  PROC DrawPart35()
    MoveL Offs(pOrigin,222.80,334.80,0.00),v40,z0,tPen\WObj:=wPaper;
    MoveL Offs(pOrigin,222.80,334.80,0.00),v40,z0,tPen\WObj:=wPaper;
    MoveL Offs(pOrigin,222.80,334.16,0.00),v40,z0,tPen\WObj:=wPaper;
    MoveL Offs(pOrigin,222.38,333.74,0.00),v40,z0,tPen\WObj:=wPaper;
    MoveL Offs(pOrigin,221.10,333.52,0.00),v40,z0,tPen\WObj:=wPaper;
    MoveL Offs(pOrigin,221.10,333.52,0.00),v40,z0,tPen\WObj:=wPaper;
    MoveL Offs(pOrigin,220.46,332.75,0.00),v40,z0,tPen\WObj:=wPaper;
    MoveL Offs(pOrigin,214.73,331.54,0.00),v40,z0,tPen\WObj:=wPaper;
    MoveL Offs(pOrigin,212.18,329.84,0.00),v40,z0,tPen\WObj:=wPaper;
    MoveL Offs(pOrigin,210.69,329.49,0.00),v40,z0,tPen\WObj:=wPaper;
    MoveL Offs(pOrigin,210.69,329.49,0.00),v40,z0,tPen\WObj:=wPaper;
    MoveL Offs(pOrigin,209.84,328.57,0.00),v40,z0,tPen\WObj:=wPaper;
    MoveL Offs(pOrigin,206.86,327.36,0.00),v40,z0,tPen\WObj:=wPaper;
    MoveL Offs(pOrigin,206.86,327.36,0.00),v40,z0,tPen\WObj:=wPaper;
    MoveL Offs(pOrigin,207.07,328.42,0.00),v40,z0,tPen\WObj:=wPaper;
    MoveL Offs(pOrigin,209.84,330.55,0.00),v40,z0,tPen\WObj:=wPaper;
    MoveL Offs(pOrigin,209.84,330.55,0.00),v40,z0,tPen\WObj:=wPaper;
    MoveL Offs(pOrigin,210.69,329.49,0.00),v40,z0,tPen\WObj:=wPaper;
    MoveL Offs(pOrigin,210.26,329.06,0.00),v40,z0,tPen\WObj:=wPaper;
    MoveL Offs(pOrigin,210.69,329.49,0.00),v40,z0,tPen\WObj:=wPaper;
    MoveL Offs(pOrigin,210.26,329.06,0.00),v40,fine,tPen\WObj:=wPaper;
    MoveL Offs(pOrigin,210.26,329.06,6.00),v60,z5,tPen\WObj:=wPaper;
    MoveL Offs(pOrigin,209.84,330.55,6.00),vTravel,z5,tPen\WObj:=wPaper;
    MoveL Offs(pOrigin,209.84,330.55,0.00),v60,z0,tPen\WObj:=wPaper;
    MoveL Offs(pOrigin,210.90,332.04,0.00),v40,z0,tPen\WObj:=wPaper;
    MoveL Offs(pOrigin,210.90,332.04,0.00),v40,z0,tPen\WObj:=wPaper;
    MoveL Offs(pOrigin,214.30,333.67,0.00),v40,z0,tPen\WObj:=wPaper;
    MoveL Offs(pOrigin,215.36,333.74,0.00),v40,z0,tPen\WObj:=wPaper;
    MoveL Offs(pOrigin,215.36,333.74,0.00),v40,z0,tPen\WObj:=wPaper;
    MoveL Offs(pOrigin,216.00,333.10,0.00),v40,z0,tPen\WObj:=wPaper;
    MoveL Offs(pOrigin,217.91,333.31,0.00),v40,z0,tPen\WObj:=wPaper;
    MoveL Offs(pOrigin,218.76,333.74,0.00),v40,z0,tPen\WObj:=wPaper;
    MoveL Offs(pOrigin,221.10,333.52,0.00),v40,z0,tPen\WObj:=wPaper;
    MoveL Offs(pOrigin,222.16,333.52,0.00),v40,z0,tPen\WObj:=wPaper;
    MoveL Offs(pOrigin,222.80,332.75,0.00),v40,z0,tPen\WObj:=wPaper;
    MoveL Offs(pOrigin,224.93,332.46,0.00),v40,z0,tPen\WObj:=wPaper;
    MoveL Offs(pOrigin,225.35,331.83,0.00),v40,fine,tPen\WObj:=wPaper;
    MoveL Offs(pOrigin,225.35,331.83,6.00),v60,z5,tPen\WObj:=wPaper;
    MoveL Offs(pOrigin,226.62,331.19,6.00),vTravel,z5,tPen\WObj:=wPaper;
    MoveL Offs(pOrigin,226.62,331.19,0.00),v60,z0,tPen\WObj:=wPaper;
    MoveL Offs(pOrigin,225.35,331.47,0.00),v40,z0,tPen\WObj:=wPaper;
    MoveL Offs(pOrigin,223.86,331.19,0.00),v40,z0,tPen\WObj:=wPaper;
    MoveL Offs(pOrigin,223.86,331.19,0.00),v40,z0,tPen\WObj:=wPaper;
    MoveL Offs(pOrigin,222.38,331.61,0.00),v40,z0,tPen\WObj:=wPaper;
    MoveL Offs(pOrigin,219.40,331.40,0.00),v40,z0,tPen\WObj:=wPaper;
    MoveL Offs(pOrigin,217.70,331.68,0.00),v40,z0,tPen\WObj:=wPaper;
    MoveL Offs(pOrigin,217.49,332.04,0.00),v40,fine,tPen\WObj:=wPaper;
    MoveL Offs(pOrigin,217.49,332.04,6.00),v60,z5,tPen\WObj:=wPaper;
    MoveL Offs(pOrigin,215.79,331.61,6.00),vTravel,z5,tPen\WObj:=wPaper;
    MoveL Offs(pOrigin,215.79,331.61,0.00),v60,z0,tPen\WObj:=wPaper;
    MoveL Offs(pOrigin,215.86,330.98,0.00),v40,z0,tPen\WObj:=wPaper;
    MoveL Offs(pOrigin,216.21,330.76,0.00),v40,z0,tPen\WObj:=wPaper;
    MoveL Offs(pOrigin,219.61,330.55,0.00),v40,z0,tPen\WObj:=wPaper;
    MoveL Offs(pOrigin,223.44,329.06,0.00),v40,z0,tPen\WObj:=wPaper;
    MoveL Offs(pOrigin,224.71,329.06,0.00),v40,z0,tPen\WObj:=wPaper;
    MoveL Offs(pOrigin,224.71,329.06,0.00),v40,z0,tPen\WObj:=wPaper;
    MoveL Offs(pOrigin,223.86,331.19,0.00),v40,fine,tPen\WObj:=wPaper;
    MoveL Offs(pOrigin,223.86,331.19,6.00),v60,z5,tPen\WObj:=wPaper;
    MoveL Offs(pOrigin,226.62,331.19,6.00),vTravel,z5,tPen\WObj:=wPaper;
    MoveL Offs(pOrigin,226.62,331.19,0.00),v60,z0,tPen\WObj:=wPaper;
    MoveL Offs(pOrigin,227.90,331.61,0.00),v40,z0,tPen\WObj:=wPaper;
    MoveL Offs(pOrigin,229.81,331.19,0.00),v40,fine,tPen\WObj:=wPaper;
    MoveL Offs(pOrigin,229.81,331.19,6.00),v60,z5,tPen\WObj:=wPaper;
    MoveL Offs(pOrigin,230.45,329.27,6.00),vTravel,z5,tPen\WObj:=wPaper;
    MoveL Offs(pOrigin,230.45,329.27,0.00),v60,z0,tPen\WObj:=wPaper;
    MoveL Offs(pOrigin,230.02,329.70,0.00),v40,z0,tPen\WObj:=wPaper;
    MoveL Offs(pOrigin,230.45,329.27,0.00),v40,fine,tPen\WObj:=wPaper;
    MoveL Offs(pOrigin,230.45,329.27,6.00),v60,z5,tPen\WObj:=wPaper;
    MoveL Offs(pOrigin,232.36,329.27,6.00),vTravel,z5,tPen\WObj:=wPaper;
    MoveL Offs(pOrigin,232.36,329.27,0.00),v60,z0,tPen\WObj:=wPaper;
    MoveL Offs(pOrigin,232.15,329.70,0.00),v40,z0,tPen\WObj:=wPaper;
    MoveL Offs(pOrigin,232.36,329.27,0.00),v40,z0,tPen\WObj:=wPaper;
    MoveL Offs(pOrigin,233.21,329.91,0.00),v40,z0,tPen\WObj:=wPaper;
    MoveL Offs(pOrigin,232.79,330.55,0.00),v40,z0,tPen\WObj:=wPaper;
    MoveL Offs(pOrigin,233.21,329.91,0.00),v40,z0,tPen\WObj:=wPaper;
    MoveL Offs(pOrigin,233.64,329.06,0.00),v40,z0,tPen\WObj:=wPaper;
    MoveL Offs(pOrigin,233.43,329.49,0.00),v40,z0,tPen\WObj:=wPaper;
    MoveL Offs(pOrigin,233.64,329.06,0.00),v40,fine,tPen\WObj:=wPaper;
    MoveL Offs(pOrigin,233.64,329.06,6.00),v60,z5,tPen\WObj:=wPaper;
    MoveL Offs(pOrigin,232.57,324.60,6.00),vTravel,z5,tPen\WObj:=wPaper;
    MoveL Offs(pOrigin,232.57,324.60,0.00),v60,z0,tPen\WObj:=wPaper;
    MoveL Offs(pOrigin,232.79,325.02,0.00),v40,z0,tPen\WObj:=wPaper;
    MoveL Offs(pOrigin,232.57,324.60,0.00),v40,fine,tPen\WObj:=wPaper;
    MoveL Offs(pOrigin,232.57,324.60,6.00),v60,z5,tPen\WObj:=wPaper;
    MoveL Offs(pOrigin,231.94,323.54,6.00),vTravel,z5,tPen\WObj:=wPaper;
    MoveL Offs(pOrigin,231.94,323.54,0.00),v60,z0,tPen\WObj:=wPaper;
    MoveL Offs(pOrigin,232.36,324.17,0.00),v40,z0,tPen\WObj:=wPaper;
    MoveL Offs(pOrigin,231.94,323.54,0.00),v40,z0,tPen\WObj:=wPaper;
    MoveL Offs(pOrigin,231.09,323.33,0.00),v40,z0,tPen\WObj:=wPaper;
    MoveL Offs(pOrigin,228.54,319.71,0.00),v40,fine,tPen\WObj:=wPaper;
    MoveL Offs(pOrigin,228.54,319.71,6.00),v60,z5,tPen\WObj:=wPaper;
    MoveL Offs(pOrigin,228.54,318.23,6.00),vTravel,z5,tPen\WObj:=wPaper;
    MoveL Offs(pOrigin,228.54,318.23,0.00),v60,z0,tPen\WObj:=wPaper;
    MoveL Offs(pOrigin,226.84,314.40,0.00),v40,z0,tPen\WObj:=wPaper;
    MoveL Offs(pOrigin,226.84,313.12,0.00),v40,z0,tPen\WObj:=wPaper;
    MoveL Offs(pOrigin,227.48,310.65,0.00),v40,z0,tPen\WObj:=wPaper;
    MoveL Offs(pOrigin,225.42,310.79,0.00),v40,z0,tPen\WObj:=wPaper;
    MoveL Offs(pOrigin,224.64,312.49,0.00),v40,z0,tPen\WObj:=wPaper;
    MoveL Offs(pOrigin,224.64,313.76,0.00),v40,z0,tPen\WObj:=wPaper;
    MoveL Offs(pOrigin,224.07,314.61,0.00),v40,z0,tPen\WObj:=wPaper;
    MoveL Offs(pOrigin,224.29,316.10,0.00),v40,fine,tPen\WObj:=wPaper;
    MoveL Offs(pOrigin,224.29,316.10,6.00),v60,z5,tPen\WObj:=wPaper;
    MoveL Offs(pOrigin,223.86,313.76,6.00),vTravel,z5,tPen\WObj:=wPaper;
    MoveL Offs(pOrigin,223.86,313.76,0.00),v60,z0,tPen\WObj:=wPaper;
    MoveL Offs(pOrigin,223.86,313.34,0.00),v40,z0,tPen\WObj:=wPaper;
    MoveL Offs(pOrigin,224.50,312.91,0.00),v40,fine,tPen\WObj:=wPaper;
    MoveL Offs(pOrigin,224.50,312.91,6.00),v60,z5,tPen\WObj:=wPaper;
    MoveL Offs(pOrigin,223.01,313.76,6.00),vTravel,z5,tPen\WObj:=wPaper;
    MoveL Offs(pOrigin,223.01,313.76,0.00),v60,z0,tPen\WObj:=wPaper;
    MoveL Offs(pOrigin,222.59,314.61,0.00),v40,z0,tPen\WObj:=wPaper;
    MoveL Offs(pOrigin,222.38,316.52,0.00),v40,z0,tPen\WObj:=wPaper;
    MoveL Offs(pOrigin,221.60,316.95,0.00),v40,z0,tPen\WObj:=wPaper;
    MoveL Offs(pOrigin,221.52,317.59,0.00),v40,z0,tPen\WObj:=wPaper;
    MoveL Offs(pOrigin,223.30,320.35,0.00),v40,z0,tPen\WObj:=wPaper;
    MoveL Offs(pOrigin,224.07,322.48,0.00),v40,z0,tPen\WObj:=wPaper;
    MoveL Offs(pOrigin,224.07,322.48,0.00),v40,z0,tPen\WObj:=wPaper;
    MoveL Offs(pOrigin,224.78,323.11,0.00),v40,z0,tPen\WObj:=wPaper;
    MoveL Offs(pOrigin,225.14,324.17,0.00),v40,z0,tPen\WObj:=wPaper;
    MoveL Offs(pOrigin,224.93,327.79,0.00),v40,z0,tPen\WObj:=wPaper;
    MoveL Offs(pOrigin,224.93,328.21,0.00),v40,z0,tPen\WObj:=wPaper;
  ENDPROC

  PROC DrawPart36()
    MoveL Offs(pOrigin,225.70,327.15,0.00),v40,z0,tPen\WObj:=wPaper;
    MoveL Offs(pOrigin,226.20,325.24,0.00),v40,z0,tPen\WObj:=wPaper;
    MoveL Offs(pOrigin,225.63,321.62,0.00),v40,z0,tPen\WObj:=wPaper;
    MoveL Offs(pOrigin,225.99,321.55,0.00),v40,z0,tPen\WObj:=wPaper;
    MoveL Offs(pOrigin,227.33,323.54,0.00),v40,z0,tPen\WObj:=wPaper;
    MoveL Offs(pOrigin,227.90,326.51,0.00),v40,z0,tPen\WObj:=wPaper;
    MoveL Offs(pOrigin,227.26,327.72,0.00),v40,z0,tPen\WObj:=wPaper;
    MoveL Offs(pOrigin,225.35,328.64,0.00),v40,z0,tPen\WObj:=wPaper;
    MoveL Offs(pOrigin,224.93,328.21,0.00),v40,fine,tPen\WObj:=wPaper;
    MoveL Offs(pOrigin,224.93,328.21,6.00),v60,z5,tPen\WObj:=wPaper;
    MoveL Offs(pOrigin,227.05,328.00,6.00),vTravel,z5,tPen\WObj:=wPaper;
    MoveL Offs(pOrigin,227.05,328.00,0.00),v60,z0,tPen\WObj:=wPaper;
    MoveL Offs(pOrigin,227.26,327.58,0.00),v40,z0,tPen\WObj:=wPaper;
    MoveL Offs(pOrigin,227.05,328.00,0.00),v40,fine,tPen\WObj:=wPaper;
    MoveL Offs(pOrigin,227.05,328.00,6.00),v60,z5,tPen\WObj:=wPaper;
    MoveL Offs(pOrigin,227.90,326.30,6.00),vTravel,z5,tPen\WObj:=wPaper;
    MoveL Offs(pOrigin,227.90,326.30,0.00),v60,z0,tPen\WObj:=wPaper;
    MoveL Offs(pOrigin,228.54,325.66,0.00),v40,z0,tPen\WObj:=wPaper;
    MoveL Offs(pOrigin,228.32,322.26,0.00),v40,fine,tPen\WObj:=wPaper;
    MoveL Offs(pOrigin,228.32,322.26,6.00),v60,z5,tPen\WObj:=wPaper;
    MoveL Offs(pOrigin,226.41,321.62,6.00),vTravel,z5,tPen\WObj:=wPaper;
    MoveL Offs(pOrigin,226.41,321.62,0.00),v60,z0,tPen\WObj:=wPaper;
    MoveL Offs(pOrigin,226.62,322.05,0.00),v40,z0,tPen\WObj:=wPaper;
    MoveL Offs(pOrigin,226.41,321.62,0.00),v40,z0,tPen\WObj:=wPaper;
    MoveL Offs(pOrigin,225.56,321.41,0.00),v40,z0,tPen\WObj:=wPaper;
    MoveL Offs(pOrigin,224.07,318.86,0.00),v40,fine,tPen\WObj:=wPaper;
    MoveL Offs(pOrigin,224.07,318.86,6.00),v60,z5,tPen\WObj:=wPaper;
    MoveL Offs(pOrigin,224.07,322.48,6.00),vTravel,z5,tPen\WObj:=wPaper;
    MoveL Offs(pOrigin,224.07,322.48,0.00),v60,z0,tPen\WObj:=wPaper;
    MoveL Offs(pOrigin,223.37,326.09,0.00),v40,z0,tPen\WObj:=wPaper;
    MoveL Offs(pOrigin,221.95,327.65,0.00),v40,z0,tPen\WObj:=wPaper;
    MoveL Offs(pOrigin,217.91,329.27,0.00),v40,z0,tPen\WObj:=wPaper;
    MoveL Offs(pOrigin,215.57,329.49,0.00),v40,z0,tPen\WObj:=wPaper;
    MoveL Offs(pOrigin,213.45,329.27,0.00),v40,z0,tPen\WObj:=wPaper;
    MoveL Offs(pOrigin,212.60,329.91,0.00),v40,fine,tPen\WObj:=wPaper;
    MoveL Offs(pOrigin,212.60,329.91,6.00),v60,z5,tPen\WObj:=wPaper;
    MoveL Offs(pOrigin,214.51,330.98,6.00),vTravel,z5,tPen\WObj:=wPaper;
    MoveL Offs(pOrigin,214.51,330.98,0.00),v60,z0,tPen\WObj:=wPaper;
    MoveL Offs(pOrigin,214.94,330.55,0.00),v40,z0,tPen\WObj:=wPaper;
    MoveL Offs(pOrigin,215.79,330.76,0.00),v40,fine,tPen\WObj:=wPaper;
    MoveL Offs(pOrigin,215.79,330.76,6.00),v60,z5,tPen\WObj:=wPaper;
    MoveL Offs(pOrigin,215.36,333.74,6.00),vTravel,z5,tPen\WObj:=wPaper;
    MoveL Offs(pOrigin,215.36,333.74,0.00),v60,z0,tPen\WObj:=wPaper;
    MoveL Offs(pOrigin,216.43,334.16,0.00),v40,z0,tPen\WObj:=wPaper;
    MoveL Offs(pOrigin,218.12,334.16,0.00),v40,z0,tPen\WObj:=wPaper;
    MoveL Offs(pOrigin,218.34,333.74,0.00),v40,fine,tPen\WObj:=wPaper;
    MoveL Offs(pOrigin,218.34,333.74,6.00),v60,z5,tPen\WObj:=wPaper;
    MoveL Offs(pOrigin,217.91,335.23,6.00),vTravel,z5,tPen\WObj:=wPaper;
    MoveL Offs(pOrigin,217.91,335.23,0.00),v60,z0,tPen\WObj:=wPaper;
    MoveL Offs(pOrigin,221.95,335.86,0.00),v40,z0,tPen\WObj:=wPaper;
    MoveL Offs(pOrigin,221.95,335.86,0.00),v40,z0,tPen\WObj:=wPaper;
    MoveL Offs(pOrigin,222.02,336.29,0.00),v40,z0,tPen\WObj:=wPaper;
    MoveL Offs(pOrigin,222.80,336.71,0.00),v40,z0,tPen\WObj:=wPaper;
    MoveL Offs(pOrigin,225.99,336.92,0.00),v40,z0,tPen\WObj:=wPaper;
    MoveL Offs(pOrigin,225.99,336.92,0.00),v40,z0,tPen\WObj:=wPaper;
    MoveL Offs(pOrigin,226.84,337.35,0.00),v40,fine,tPen\WObj:=wPaper;
    MoveL Offs(pOrigin,226.84,337.35,6.00),v60,z5,tPen\WObj:=wPaper;
    MoveL Offs(pOrigin,224.71,335.86,6.00),vTravel,z5,tPen\WObj:=wPaper;
    MoveL Offs(pOrigin,224.71,335.86,0.00),v60,z0,tPen\WObj:=wPaper;
    MoveL Offs(pOrigin,222.59,335.65,0.00),v40,fine,tPen\WObj:=wPaper;
    MoveL Offs(pOrigin,222.59,335.65,6.00),v60,z5,tPen\WObj:=wPaper;
    MoveL Offs(pOrigin,226.62,331.19,6.00),vTravel,z5,tPen\WObj:=wPaper;
    MoveL Offs(pOrigin,226.62,331.19,0.00),v60,z0,tPen\WObj:=wPaper;
    MoveL Offs(pOrigin,229.53,328.64,0.00),v40,z0,tPen\WObj:=wPaper;
    MoveL Offs(pOrigin,230.02,327.36,0.00),v40,z0,tPen\WObj:=wPaper;
    MoveL Offs(pOrigin,230.02,325.02,0.00),v40,z0,tPen\WObj:=wPaper;
    MoveL Offs(pOrigin,229.10,322.55,0.00),v40,z0,tPen\WObj:=wPaper;
    MoveL Offs(pOrigin,228.32,322.05,0.00),v40,z0,tPen\WObj:=wPaper;
    MoveL Offs(pOrigin,226.13,318.65,0.00),v40,z0,tPen\WObj:=wPaper;
    MoveL Offs(pOrigin,225.70,316.95,0.00),v40,z0,tPen\WObj:=wPaper;
    MoveL Offs(pOrigin,226.41,316.31,0.00),v40,z0,tPen\WObj:=wPaper;
    MoveL Offs(pOrigin,225.99,315.25,0.00),v40,z0,tPen\WObj:=wPaper;
    MoveL Offs(pOrigin,226.20,314.61,0.00),v40,z0,tPen\WObj:=wPaper;
    MoveL Offs(pOrigin,227.05,314.61,0.00),v40,z0,tPen\WObj:=wPaper;
    MoveL Offs(pOrigin,228.18,312.13,0.00),v40,z0,tPen\WObj:=wPaper;
    MoveL Offs(pOrigin,228.96,311.85,0.00),v40,z0,tPen\WObj:=wPaper;
    MoveL Offs(pOrigin,228.96,311.85,0.00),v40,z0,tPen\WObj:=wPaper;
    MoveL Offs(pOrigin,229.39,311.00,0.00),v40,z0,tPen\WObj:=wPaper;
    MoveL Offs(pOrigin,229.39,311.00,0.00),v40,z0,tPen\WObj:=wPaper;
    MoveL Offs(pOrigin,228.54,310.15,0.00),v40,z0,tPen\WObj:=wPaper;
    MoveL Offs(pOrigin,227.69,310.58,0.00),v40,z0,tPen\WObj:=wPaper;
    MoveL Offs(pOrigin,228.75,310.15,0.00),v40,z0,tPen\WObj:=wPaper;
    MoveL Offs(pOrigin,229.39,311.00,0.00),v40,z0,tPen\WObj:=wPaper;
    MoveL Offs(pOrigin,229.39,311.00,0.00),v40,z0,tPen\WObj:=wPaper;
    MoveL Offs(pOrigin,230.02,311.00,0.00),v40,z0,tPen\WObj:=wPaper;
    MoveL Offs(pOrigin,230.88,312.06,0.00),v40,z0,tPen\WObj:=wPaper;
    MoveL Offs(pOrigin,230.88,311.64,0.00),v40,z0,tPen\WObj:=wPaper;
    MoveL Offs(pOrigin,232.57,310.58,0.00),v40,z0,tPen\WObj:=wPaper;
    MoveL Offs(pOrigin,233.43,311.00,0.00),v40,fine,tPen\WObj:=wPaper;
    MoveL Offs(pOrigin,233.43,311.00,6.00),v60,z5,tPen\WObj:=wPaper;
    MoveL Offs(pOrigin,235.55,311.42,6.00),vTravel,z5,tPen\WObj:=wPaper;
    MoveL Offs(pOrigin,235.55,311.42,0.00),v60,z0,tPen\WObj:=wPaper;
    MoveL Offs(pOrigin,234.98,311.71,0.00),v40,z0,tPen\WObj:=wPaper;
    MoveL Offs(pOrigin,234.70,312.49,0.00),v40,z0,tPen\WObj:=wPaper;
    MoveL Offs(pOrigin,234.70,315.46,0.00),v40,z0,tPen\WObj:=wPaper;
    MoveL Offs(pOrigin,235.12,317.38,0.00),v40,fine,tPen\WObj:=wPaper;
    MoveL Offs(pOrigin,235.12,317.38,6.00),v60,z5,tPen\WObj:=wPaper;
    MoveL Offs(pOrigin,232.79,318.44,6.00),vTravel,z5,tPen\WObj:=wPaper;
    MoveL Offs(pOrigin,232.79,318.44,0.00),v60,z0,tPen\WObj:=wPaper;
    MoveL Offs(pOrigin,234.27,320.14,0.00),v40,z0,tPen\WObj:=wPaper;
    MoveL Offs(pOrigin,234.27,320.56,0.00),v40,fine,tPen\WObj:=wPaper;
    MoveL Offs(pOrigin,234.27,320.56,6.00),v60,z5,tPen\WObj:=wPaper;
    MoveL Offs(pOrigin,235.55,321.41,6.00),vTravel,z5,tPen\WObj:=wPaper;
    MoveL Offs(pOrigin,235.55,321.41,0.00),v60,z0,tPen\WObj:=wPaper;
    MoveL Offs(pOrigin,234.91,320.70,0.00),v40,z0,tPen\WObj:=wPaper;
    MoveL Offs(pOrigin,234.35,320.77,0.00),v40,z0,tPen\WObj:=wPaper;
    MoveL Offs(pOrigin,234.70,321.84,0.00),v40,z0,tPen\WObj:=wPaper;
    MoveL Offs(pOrigin,235.55,322.05,0.00),v40,z0,tPen\WObj:=wPaper;
    MoveL Offs(pOrigin,235.55,322.05,0.00),v40,z0,tPen\WObj:=wPaper;
    MoveL Offs(pOrigin,237.89,325.66,0.00),v40,fine,tPen\WObj:=wPaper;
    MoveL Offs(pOrigin,237.89,325.66,6.00),v60,z5,tPen\WObj:=wPaper;
    MoveL Offs(pOrigin,239.80,326.73,6.00),vTravel,z5,tPen\WObj:=wPaper;
    MoveL Offs(pOrigin,239.80,326.73,0.00),v60,z0,tPen\WObj:=wPaper;
    MoveL Offs(pOrigin,239.16,327.15,0.00),v40,z0,tPen\WObj:=wPaper;
    MoveL Offs(pOrigin,239.38,328.00,0.00),v40,fine,tPen\WObj:=wPaper;
    MoveL Offs(pOrigin,239.38,328.00,6.00),v60,z5,tPen\WObj:=wPaper;
    MoveL Offs(pOrigin,242.14,324.60,6.00),vTravel,z5,tPen\WObj:=wPaper;
    MoveL Offs(pOrigin,242.14,324.60,0.00),v60,z0,tPen\WObj:=wPaper;
    MoveL Offs(pOrigin,242.56,325.24,0.00),v40,z0,tPen\WObj:=wPaper;
    MoveL Offs(pOrigin,242.14,324.60,0.00),v40,fine,tPen\WObj:=wPaper;
  ENDPROC

  PROC DrawPart37()
    MoveL Offs(pOrigin,242.14,324.60,6.00),v60,z5,tPen\WObj:=wPaper;
    MoveL Offs(pOrigin,239.59,323.11,6.00),vTravel,z5,tPen\WObj:=wPaper;
    MoveL Offs(pOrigin,239.59,323.11,0.00),v60,z0,tPen\WObj:=wPaper;
    MoveL Offs(pOrigin,237.04,320.77,0.00),v40,z0,tPen\WObj:=wPaper;
    MoveL Offs(pOrigin,237.04,320.77,0.00),v40,z0,tPen\WObj:=wPaper;
    MoveL Offs(pOrigin,235.76,321.41,0.00),v40,z0,tPen\WObj:=wPaper;
    MoveL Offs(pOrigin,235.55,322.05,0.00),v40,fine,tPen\WObj:=wPaper;
    MoveL Offs(pOrigin,235.55,322.05,6.00),v60,z5,tPen\WObj:=wPaper;
    MoveL Offs(pOrigin,237.04,320.77,6.00),vTravel,z5,tPen\WObj:=wPaper;
    MoveL Offs(pOrigin,237.04,320.77,0.00),v60,z0,tPen\WObj:=wPaper;
    MoveL Offs(pOrigin,235.34,317.80,0.00),v40,z0,tPen\WObj:=wPaper;
    MoveL Offs(pOrigin,234.20,316.95,0.00),v40,z0,tPen\WObj:=wPaper;
    MoveL Offs(pOrigin,233.64,315.25,0.00),v40,z0,tPen\WObj:=wPaper;
    MoveL Offs(pOrigin,233.43,313.34,0.00),v40,z0,tPen\WObj:=wPaper;
    MoveL Offs(pOrigin,233.64,312.49,0.00),v40,z0,tPen\WObj:=wPaper;
    MoveL Offs(pOrigin,233.21,311.99,0.00),v40,z0,tPen\WObj:=wPaper;
    MoveL Offs(pOrigin,232.57,313.12,0.00),v40,z0,tPen\WObj:=wPaper;
    MoveL Offs(pOrigin,232.57,315.25,0.00),v40,z0,tPen\WObj:=wPaper;
    MoveL Offs(pOrigin,233.21,317.16,0.00),v40,z0,tPen\WObj:=wPaper;
    MoveL Offs(pOrigin,232.79,318.44,0.00),v40,z0,tPen\WObj:=wPaper;
    MoveL Offs(pOrigin,232.79,318.44,0.00),v40,z0,tPen\WObj:=wPaper;
    MoveL Offs(pOrigin,232.15,317.80,0.00),v40,z0,tPen\WObj:=wPaper;
    MoveL Offs(pOrigin,232.15,317.80,0.00),v40,z0,tPen\WObj:=wPaper;
    MoveL Offs(pOrigin,231.51,314.61,0.00),v40,z0,tPen\WObj:=wPaper;
    MoveL Offs(pOrigin,230.88,313.76,0.00),v40,z0,tPen\WObj:=wPaper;
    MoveL Offs(pOrigin,230.88,313.76,0.00),v40,z0,tPen\WObj:=wPaper;
    MoveL Offs(pOrigin,230.80,312.27,0.00),v40,z0,tPen\WObj:=wPaper;
    MoveL Offs(pOrigin,229.25,312.91,0.00),v40,z0,tPen\WObj:=wPaper;
    MoveL Offs(pOrigin,228.96,316.74,0.00),v40,z0,tPen\WObj:=wPaper;
    MoveL Offs(pOrigin,228.96,316.74,0.00),v40,z0,tPen\WObj:=wPaper;
    MoveL Offs(pOrigin,229.81,316.74,0.00),v40,z0,tPen\WObj:=wPaper;
    MoveL Offs(pOrigin,230.66,318.01,0.00),v40,z0,tPen\WObj:=wPaper;
    MoveL Offs(pOrigin,230.66,318.01,0.00),v40,z0,tPen\WObj:=wPaper;
    MoveL Offs(pOrigin,231.09,319.08,0.00),v40,z0,tPen\WObj:=wPaper;
    MoveL Offs(pOrigin,231.09,319.08,0.00),v40,z0,tPen\WObj:=wPaper;
    MoveL Offs(pOrigin,231.16,320.56,0.00),v40,z0,tPen\WObj:=wPaper;
    MoveL Offs(pOrigin,233.43,323.11,0.00),v40,z0,tPen\WObj:=wPaper;
    MoveL Offs(pOrigin,233.21,322.69,0.00),v40,z0,tPen\WObj:=wPaper;
    MoveL Offs(pOrigin,233.43,323.11,0.00),v40,z0,tPen\WObj:=wPaper;
    MoveL Offs(pOrigin,233.21,322.69,0.00),v40,fine,tPen\WObj:=wPaper;
    MoveL Offs(pOrigin,233.21,322.69,6.00),v60,z5,tPen\WObj:=wPaper;
    MoveL Offs(pOrigin,231.09,319.08,6.00),vTravel,z5,tPen\WObj:=wPaper;
    MoveL Offs(pOrigin,231.09,319.08,0.00),v60,z0,tPen\WObj:=wPaper;
    MoveL Offs(pOrigin,231.94,319.08,0.00),v40,z0,tPen\WObj:=wPaper;
    MoveL Offs(pOrigin,232.57,318.44,0.00),v40,z0,tPen\WObj:=wPaper;
    MoveL Offs(pOrigin,232.57,318.44,0.00),v40,z0,tPen\WObj:=wPaper;
    MoveL Offs(pOrigin,231.94,317.80,0.00),v40,z0,tPen\WObj:=wPaper;
    MoveL Offs(pOrigin,231.30,317.80,0.00),v40,z0,tPen\WObj:=wPaper;
    MoveL Offs(pOrigin,231.30,317.80,0.00),v40,z0,tPen\WObj:=wPaper;
    MoveL Offs(pOrigin,231.09,316.52,0.00),v40,z0,tPen\WObj:=wPaper;
    MoveL Offs(pOrigin,230.45,316.10,0.00),v40,z0,tPen\WObj:=wPaper;
    MoveL Offs(pOrigin,230.45,316.10,0.00),v40,z0,tPen\WObj:=wPaper;
    MoveL Offs(pOrigin,230.45,314.19,0.00),v40,z0,tPen\WObj:=wPaper;
    MoveL Offs(pOrigin,230.88,313.76,0.00),v40,fine,tPen\WObj:=wPaper;
    MoveL Offs(pOrigin,230.88,313.76,6.00),v60,z5,tPen\WObj:=wPaper;
    MoveL Offs(pOrigin,230.88,311.64,6.00),vTravel,z5,tPen\WObj:=wPaper;
    MoveL Offs(pOrigin,230.88,311.64,0.00),v60,z0,tPen\WObj:=wPaper;
    MoveL Offs(pOrigin,230.24,311.00,0.00),v40,fine,tPen\WObj:=wPaper;
    MoveL Offs(pOrigin,230.24,311.00,6.00),v60,z5,tPen\WObj:=wPaper;
    MoveL Offs(pOrigin,226.84,309.30,6.00),vTravel,z5,tPen\WObj:=wPaper;
    MoveL Offs(pOrigin,226.84,309.30,0.00),v60,z0,tPen\WObj:=wPaper;
    MoveL Offs(pOrigin,225.56,310.36,0.00),v40,z0,tPen\WObj:=wPaper;
    MoveL Offs(pOrigin,224.07,310.15,0.00),v40,z0,tPen\WObj:=wPaper;
    MoveL Offs(pOrigin,222.59,310.50,0.00),v40,z0,tPen\WObj:=wPaper;
    MoveL Offs(pOrigin,222.45,309.51,0.00),v40,z0,tPen\WObj:=wPaper;
    MoveL Offs(pOrigin,223.86,308.88,0.00),v40,fine,tPen\WObj:=wPaper;
    MoveL Offs(pOrigin,223.86,308.88,6.00),v60,z5,tPen\WObj:=wPaper;
    MoveL Offs(pOrigin,222.38,309.30,6.00),vTravel,z5,tPen\WObj:=wPaper;
    MoveL Offs(pOrigin,222.38,309.30,0.00),v60,z0,tPen\WObj:=wPaper;
    MoveL Offs(pOrigin,221.31,308.66,0.00),v40,z0,tPen\WObj:=wPaper;
    MoveL Offs(pOrigin,220.89,308.88,0.00),v40,z0,tPen\WObj:=wPaper;
    MoveL Offs(pOrigin,220.46,308.24,0.00),v40,z0,tPen\WObj:=wPaper;
    MoveL Offs(pOrigin,220.46,308.24,0.00),v40,z0,tPen\WObj:=wPaper;
    MoveL Offs(pOrigin,220.68,308.24,0.00),v40,z0,tPen\WObj:=wPaper;
    MoveL Offs(pOrigin,220.04,307.39,0.00),v40,z0,tPen\WObj:=wPaper;
    MoveL Offs(pOrigin,218.76,307.39,0.00),v40,z0,tPen\WObj:=wPaper;
    MoveL Offs(pOrigin,218.76,307.39,0.00),v40,z0,tPen\WObj:=wPaper;
    MoveL Offs(pOrigin,218.12,306.61,0.00),v40,z0,tPen\WObj:=wPaper;
    MoveL Offs(pOrigin,217.06,306.61,0.00),v40,z0,tPen\WObj:=wPaper;
    MoveL Offs(pOrigin,217.49,308.02,0.00),v40,z0,tPen\WObj:=wPaper;
    MoveL Offs(pOrigin,217.49,308.02,0.00),v40,z0,tPen\WObj:=wPaper;
    MoveL Offs(pOrigin,218.34,308.02,0.00),v40,z0,tPen\WObj:=wPaper;
    MoveL Offs(pOrigin,218.76,308.45,0.00),v40,z0,tPen\WObj:=wPaper;
    MoveL Offs(pOrigin,218.76,309.51,0.00),v40,z0,tPen\WObj:=wPaper;
    MoveL Offs(pOrigin,218.76,309.51,0.00),v40,z0,tPen\WObj:=wPaper;
    MoveL Offs(pOrigin,220.68,309.09,0.00),v40,z0,tPen\WObj:=wPaper;
    MoveL Offs(pOrigin,220.46,308.24,0.00),v40,z0,tPen\WObj:=wPaper;
    MoveL Offs(pOrigin,218.76,308.24,0.00),v40,fine,tPen\WObj:=wPaper;
    MoveL Offs(pOrigin,218.76,308.24,6.00),v60,z5,tPen\WObj:=wPaper;
    MoveL Offs(pOrigin,217.49,308.02,6.00),vTravel,z5,tPen\WObj:=wPaper;
    MoveL Offs(pOrigin,217.49,308.02,0.00),v60,z0,tPen\WObj:=wPaper;
    MoveL Offs(pOrigin,215.79,308.45,0.00),v40,z0,tPen\WObj:=wPaper;
    MoveL Offs(pOrigin,214.94,309.16,0.00),v40,z0,tPen\WObj:=wPaper;
    MoveL Offs(pOrigin,214.51,308.88,0.00),v40,z0,tPen\WObj:=wPaper;
    MoveL Offs(pOrigin,214.73,309.30,0.00),v40,z0,tPen\WObj:=wPaper;
    MoveL Offs(pOrigin,214.09,308.52,0.00),v40,z0,tPen\WObj:=wPaper;
    MoveL Offs(pOrigin,213.45,308.38,0.00),v40,z0,tPen\WObj:=wPaper;
    MoveL Offs(pOrigin,210.26,309.94,0.00),v40,z0,tPen\WObj:=wPaper;
    MoveL Offs(pOrigin,210.26,309.94,0.00),v40,z0,tPen\WObj:=wPaper;
    MoveL Offs(pOrigin,209.98,310.72,0.00),v40,z0,tPen\WObj:=wPaper;
    MoveL Offs(pOrigin,207.50,312.27,0.00),v40,z0,tPen\WObj:=wPaper;
    MoveL Offs(pOrigin,206.65,313.55,0.00),v40,z0,tPen\WObj:=wPaper;
    MoveL Offs(pOrigin,206.65,313.55,0.00),v40,z0,tPen\WObj:=wPaper;
    MoveL Offs(pOrigin,206.44,313.98,0.00),v40,z0,tPen\WObj:=wPaper;
    MoveL Offs(pOrigin,205.16,314.40,0.00),v40,z0,tPen\WObj:=wPaper;
    MoveL Offs(pOrigin,205.16,314.40,0.00),v40,z0,tPen\WObj:=wPaper;
    MoveL Offs(pOrigin,204.31,314.19,0.00),v40,z0,tPen\WObj:=wPaper;
    MoveL Offs(pOrigin,203.89,314.61,0.00),v40,z0,tPen\WObj:=wPaper;
    MoveL Offs(pOrigin,203.89,314.61,0.00),v40,z0,tPen\WObj:=wPaper;
    MoveL Offs(pOrigin,202.19,314.40,0.00),v40,z0,tPen\WObj:=wPaper;
    MoveL Offs(pOrigin,201.76,315.04,0.00),v40,fine,tPen\WObj:=wPaper;
    MoveL Offs(pOrigin,201.76,315.04,6.00),v60,z5,tPen\WObj:=wPaper;
    MoveL Offs(pOrigin,203.04,315.67,6.00),vTravel,z5,tPen\WObj:=wPaper;
    MoveL Offs(pOrigin,203.04,315.67,0.00),v60,z0,tPen\WObj:=wPaper;
    MoveL Offs(pOrigin,203.46,316.10,0.00),v40,z0,tPen\WObj:=wPaper;
    MoveL Offs(pOrigin,205.38,316.10,0.00),v40,z0,tPen\WObj:=wPaper;
    MoveL Offs(pOrigin,205.38,316.10,0.00),v40,z0,tPen\WObj:=wPaper;
    MoveL Offs(pOrigin,205.59,316.88,0.00),v40,z0,tPen\WObj:=wPaper;
    MoveL Offs(pOrigin,206.86,316.95,0.00),v40,z0,tPen\WObj:=wPaper;
    MoveL Offs(pOrigin,208.35,316.52,0.00),v40,z0,tPen\WObj:=wPaper;
  ENDPROC

  PROC DrawPart38()
    MoveL Offs(pOrigin,209.41,316.60,0.00),v40,z0,tPen\WObj:=wPaper;
    MoveL Offs(pOrigin,210.69,315.75,0.00),v40,z0,tPen\WObj:=wPaper;
    MoveL Offs(pOrigin,211.32,315.67,0.00),v40,z0,tPen\WObj:=wPaper;
    MoveL Offs(pOrigin,211.32,315.67,0.00),v40,z0,tPen\WObj:=wPaper;
    MoveL Offs(pOrigin,211.96,315.89,0.00),v40,z0,tPen\WObj:=wPaper;
    MoveL Offs(pOrigin,212.18,316.74,0.00),v40,z0,tPen\WObj:=wPaper;
    MoveL Offs(pOrigin,211.68,318.65,0.00),v40,z0,tPen\WObj:=wPaper;
    MoveL Offs(pOrigin,210.90,319.71,0.00),v40,z0,tPen\WObj:=wPaper;
    MoveL Offs(pOrigin,210.90,319.71,0.00),v40,z0,tPen\WObj:=wPaper;
    MoveL Offs(pOrigin,211.96,320.99,0.00),v40,z0,tPen\WObj:=wPaper;
    MoveL Offs(pOrigin,211.96,320.99,0.00),v40,z0,tPen\WObj:=wPaper;
    MoveL Offs(pOrigin,213.10,320.35,0.00),v40,z0,tPen\WObj:=wPaper;
    MoveL Offs(pOrigin,214.37,315.04,0.00),v40,z0,tPen\WObj:=wPaper;
    MoveL Offs(pOrigin,215.15,314.61,0.00),v40,z0,tPen\WObj:=wPaper;
    MoveL Offs(pOrigin,215.15,314.61,0.00),v40,z0,tPen\WObj:=wPaper;
    MoveL Offs(pOrigin,214.94,316.10,0.00),v40,z0,tPen\WObj:=wPaper;
    MoveL Offs(pOrigin,215.15,320.56,0.00),v40,z0,tPen\WObj:=wPaper;
    MoveL Offs(pOrigin,214.65,321.98,0.00),v40,z0,tPen\WObj:=wPaper;
    MoveL Offs(pOrigin,213.66,322.69,0.00),v40,fine,tPen\WObj:=wPaper;
    MoveL Offs(pOrigin,213.66,322.69,6.00),v60,z5,tPen\WObj:=wPaper;
    MoveL Offs(pOrigin,211.96,320.99,6.00),vTravel,z5,tPen\WObj:=wPaper;
    MoveL Offs(pOrigin,211.96,320.99,0.00),v60,z0,tPen\WObj:=wPaper;
    MoveL Offs(pOrigin,211.75,321.34,0.00),v40,z0,tPen\WObj:=wPaper;
    MoveL Offs(pOrigin,208.77,322.69,0.00),v40,z0,tPen\WObj:=wPaper;
    MoveL Offs(pOrigin,205.16,322.90,0.00),v40,fine,tPen\WObj:=wPaper;
    MoveL Offs(pOrigin,205.16,322.90,6.00),v60,z5,tPen\WObj:=wPaper;
    MoveL Offs(pOrigin,205.38,321.62,6.00),vTravel,z5,tPen\WObj:=wPaper;
    MoveL Offs(pOrigin,205.38,321.62,0.00),v60,z0,tPen\WObj:=wPaper;
    MoveL Offs(pOrigin,204.10,321.13,0.00),v40,z0,tPen\WObj:=wPaper;
    MoveL Offs(pOrigin,202.61,321.41,0.00),v40,z0,tPen\WObj:=wPaper;
    MoveL Offs(pOrigin,202.61,321.41,0.00),v40,z0,tPen\WObj:=wPaper;
    MoveL Offs(pOrigin,203.25,322.33,0.00),v40,z0,tPen\WObj:=wPaper;
    MoveL Offs(pOrigin,206.23,323.75,0.00),v40,z0,tPen\WObj:=wPaper;
    MoveL Offs(pOrigin,206.23,323.75,0.00),v40,z0,tPen\WObj:=wPaper;
    MoveL Offs(pOrigin,207.29,323.96,0.00),v40,z0,tPen\WObj:=wPaper;
    MoveL Offs(pOrigin,207.29,323.96,0.00),v40,z0,tPen\WObj:=wPaper;
    MoveL Offs(pOrigin,210.05,323.96,0.00),v40,z0,tPen\WObj:=wPaper;
    MoveL Offs(pOrigin,213.24,322.69,0.00),v40,z0,tPen\WObj:=wPaper;
    MoveL Offs(pOrigin,213.52,322.90,0.00),v40,z0,tPen\WObj:=wPaper;
    MoveL Offs(pOrigin,213.31,323.54,0.00),v40,z0,tPen\WObj:=wPaper;
    MoveL Offs(pOrigin,210.48,324.81,0.00),v40,z0,tPen\WObj:=wPaper;
    MoveL Offs(pOrigin,208.35,325.02,0.00),v40,z0,tPen\WObj:=wPaper;
    MoveL Offs(pOrigin,207.29,324.81,0.00),v40,z0,tPen\WObj:=wPaper;
    MoveL Offs(pOrigin,209.84,326.23,0.00),v40,z0,tPen\WObj:=wPaper;
    MoveL Offs(pOrigin,211.32,326.37,0.00),v40,z0,tPen\WObj:=wPaper;
    MoveL Offs(pOrigin,212.39,327.15,0.00),v40,z0,tPen\WObj:=wPaper;
    MoveL Offs(pOrigin,215.57,327.36,0.00),v40,z0,tPen\WObj:=wPaper;
    MoveL Offs(pOrigin,218.34,326.73,0.00),v40,z0,tPen\WObj:=wPaper;
    MoveL Offs(pOrigin,218.34,326.73,0.00),v40,z0,tPen\WObj:=wPaper;
    MoveL Offs(pOrigin,218.98,323.54,0.00),v40,z0,tPen\WObj:=wPaper;
    MoveL Offs(pOrigin,218.98,321.84,0.00),v40,z0,tPen\WObj:=wPaper;
    MoveL Offs(pOrigin,218.98,321.84,0.00),v40,z0,tPen\WObj:=wPaper;
    MoveL Offs(pOrigin,219.40,321.62,0.00),v40,z0,tPen\WObj:=wPaper;
    MoveL Offs(pOrigin,219.61,320.99,0.00),v40,z0,tPen\WObj:=wPaper;
    MoveL Offs(pOrigin,219.61,320.99,0.00),v40,z0,tPen\WObj:=wPaper;
    MoveL Offs(pOrigin,219.19,318.23,0.00),v40,z0,tPen\WObj:=wPaper;
    MoveL Offs(pOrigin,220.04,317.59,0.00),v40,z0,tPen\WObj:=wPaper;
    MoveL Offs(pOrigin,220.18,313.98,0.00),v40,z0,tPen\WObj:=wPaper;
    MoveL Offs(pOrigin,219.40,313.41,0.00),v40,z0,tPen\WObj:=wPaper;
    MoveL Offs(pOrigin,217.06,313.83,0.00),v40,z0,tPen\WObj:=wPaper;
    MoveL Offs(pOrigin,216.64,314.40,0.00),v40,z0,tPen\WObj:=wPaper;
    MoveL Offs(pOrigin,216.64,315.25,0.00),v40,z0,tPen\WObj:=wPaper;
    MoveL Offs(pOrigin,217.27,315.67,0.00),v40,z0,tPen\WObj:=wPaper;
    MoveL Offs(pOrigin,217.27,315.67,0.00),v40,z0,tPen\WObj:=wPaper;
    MoveL Offs(pOrigin,217.06,316.74,0.00),v40,z0,tPen\WObj:=wPaper;
    MoveL Offs(pOrigin,217.49,320.35,0.00),v40,z0,tPen\WObj:=wPaper;
    MoveL Offs(pOrigin,217.49,320.35,0.00),v40,z0,tPen\WObj:=wPaper;
    MoveL Offs(pOrigin,218.12,320.35,0.00),v40,z0,tPen\WObj:=wPaper;
    MoveL Offs(pOrigin,218.55,320.77,0.00),v40,z0,tPen\WObj:=wPaper;
    MoveL Offs(pOrigin,218.55,321.41,0.00),v40,z0,tPen\WObj:=wPaper;
    MoveL Offs(pOrigin,218.98,321.84,0.00),v40,z0,tPen\WObj:=wPaper;
    MoveL Offs(pOrigin,219.61,320.99,0.00),v40,z0,tPen\WObj:=wPaper;
    MoveL Offs(pOrigin,220.46,321.84,0.00),v40,z0,tPen\WObj:=wPaper;
    MoveL Offs(pOrigin,220.46,321.84,0.00),v40,z0,tPen\WObj:=wPaper;
    MoveL Offs(pOrigin,221.52,321.84,0.00),v40,z0,tPen\WObj:=wPaper;
    MoveL Offs(pOrigin,221.31,321.41,0.00),v40,z0,tPen\WObj:=wPaper;
    MoveL Offs(pOrigin,221.52,321.84,0.00),v40,z0,tPen\WObj:=wPaper;
    MoveL Offs(pOrigin,221.31,321.41,0.00),v40,z0,tPen\WObj:=wPaper;
    MoveL Offs(pOrigin,220.46,321.84,0.00),v40,z0,tPen\WObj:=wPaper;
    MoveL Offs(pOrigin,220.68,323.96,0.00),v40,fine,tPen\WObj:=wPaper;
    MoveL Offs(pOrigin,220.68,323.96,6.00),v60,z5,tPen\WObj:=wPaper;
    MoveL Offs(pOrigin,220.68,325.24,6.00),vTravel,z5,tPen\WObj:=wPaper;
    MoveL Offs(pOrigin,220.68,325.24,0.00),v60,z0,tPen\WObj:=wPaper;
    MoveL Offs(pOrigin,221.95,325.66,0.00),v40,z0,tPen\WObj:=wPaper;
    MoveL Offs(pOrigin,221.95,325.66,0.00),v40,z0,tPen\WObj:=wPaper;
    MoveL Offs(pOrigin,222.59,325.24,0.00),v40,z0,tPen\WObj:=wPaper;
    MoveL Offs(pOrigin,222.59,323.11,0.00),v40,z0,tPen\WObj:=wPaper;
    MoveL Offs(pOrigin,221.95,322.26,0.00),v40,z0,tPen\WObj:=wPaper;
    MoveL Offs(pOrigin,221.95,322.26,0.00),v40,z0,tPen\WObj:=wPaper;
    MoveL Offs(pOrigin,220.75,324.17,0.00),v40,z0,tPen\WObj:=wPaper;
    MoveL Offs(pOrigin,220.68,325.24,0.00),v40,z0,tPen\WObj:=wPaper;
    MoveL Offs(pOrigin,220.68,325.24,0.00),v40,z0,tPen\WObj:=wPaper;
    MoveL Offs(pOrigin,220.25,325.24,0.00),v40,z0,tPen\WObj:=wPaper;
    MoveL Offs(pOrigin,220.04,325.88,0.00),v40,z0,tPen\WObj:=wPaper;
    MoveL Offs(pOrigin,218.76,326.73,0.00),v40,z0,tPen\WObj:=wPaper;
    MoveL Offs(pOrigin,218.76,326.73,0.00),v40,z0,tPen\WObj:=wPaper;
    MoveL Offs(pOrigin,219.61,327.36,0.00),v40,z0,tPen\WObj:=wPaper;
    MoveL Offs(pOrigin,220.68,327.29,0.00),v40,z0,tPen\WObj:=wPaper;
    MoveL Offs(pOrigin,221.88,326.30,0.00),v40,z0,tPen\WObj:=wPaper;
    MoveL Offs(pOrigin,221.95,325.66,0.00),v40,z0,tPen\WObj:=wPaper;
    MoveL Offs(pOrigin,221.74,326.30,0.00),v40,z0,tPen\WObj:=wPaper;
    MoveL Offs(pOrigin,221.52,326.73,0.00),v40,z0,tPen\WObj:=wPaper;
    MoveL Offs(pOrigin,221.74,326.30,0.00),v40,fine,tPen\WObj:=wPaper;
    MoveL Offs(pOrigin,221.74,326.30,6.00),v60,z5,tPen\WObj:=wPaper;
    MoveL Offs(pOrigin,222.59,327.15,6.00),vTravel,z5,tPen\WObj:=wPaper;
    MoveL Offs(pOrigin,222.59,327.15,0.00),v60,z0,tPen\WObj:=wPaper;
    MoveL Offs(pOrigin,222.80,326.73,0.00),v40,z0,tPen\WObj:=wPaper;
    MoveL Offs(pOrigin,222.59,327.15,0.00),v40,z0,tPen\WObj:=wPaper;
    MoveL Offs(pOrigin,221.95,327.79,0.00),v40,z0,tPen\WObj:=wPaper;
    MoveL Offs(pOrigin,222.16,327.36,0.00),v40,z0,tPen\WObj:=wPaper;
    MoveL Offs(pOrigin,221.95,327.79,0.00),v40,fine,tPen\WObj:=wPaper;
    MoveL Offs(pOrigin,221.95,327.79,6.00),v60,z5,tPen\WObj:=wPaper;
    MoveL Offs(pOrigin,220.68,328.42,6.00),vTravel,z5,tPen\WObj:=wPaper;
    MoveL Offs(pOrigin,220.68,328.42,0.00),v60,z0,tPen\WObj:=wPaper;
    MoveL Offs(pOrigin,221.10,328.21,0.00),v40,z0,tPen\WObj:=wPaper;
    MoveL Offs(pOrigin,220.68,328.42,0.00),v40,fine,tPen\WObj:=wPaper;
    MoveL Offs(pOrigin,220.68,328.42,6.00),v60,z5,tPen\WObj:=wPaper;
    MoveL Offs(pOrigin,219.19,327.36,6.00),vTravel,z5,tPen\WObj:=wPaper;
    MoveL Offs(pOrigin,219.19,327.36,0.00),v60,z0,tPen\WObj:=wPaper;
    MoveL Offs(pOrigin,218.34,326.73,0.00),v40,fine,tPen\WObj:=wPaper;
  ENDPROC

  PROC DrawPart39()
    MoveL Offs(pOrigin,218.34,326.73,6.00),v60,z5,tPen\WObj:=wPaper;
    MoveL Offs(pOrigin,215.79,324.17,6.00),vTravel,z5,tPen\WObj:=wPaper;
    MoveL Offs(pOrigin,215.79,324.17,0.00),v60,z0,tPen\WObj:=wPaper;
    MoveL Offs(pOrigin,214.30,325.59,0.00),v40,z0,tPen\WObj:=wPaper;
    MoveL Offs(pOrigin,211.96,326.16,0.00),v40,z0,tPen\WObj:=wPaper;
    MoveL Offs(pOrigin,211.75,326.51,0.00),v40,fine,tPen\WObj:=wPaper;
    MoveL Offs(pOrigin,211.75,326.51,6.00),v60,z5,tPen\WObj:=wPaper;
    MoveL Offs(pOrigin,209.41,325.66,6.00),vTravel,z5,tPen\WObj:=wPaper;
    MoveL Offs(pOrigin,209.41,325.66,0.00),v60,z0,tPen\WObj:=wPaper;
    MoveL Offs(pOrigin,209.84,326.09,0.00),v40,z0,tPen\WObj:=wPaper;
    MoveL Offs(pOrigin,209.41,325.66,0.00),v40,fine,tPen\WObj:=wPaper;
    MoveL Offs(pOrigin,209.41,325.66,6.00),v60,z5,tPen\WObj:=wPaper;
    MoveL Offs(pOrigin,207.29,324.81,6.00),vTravel,z5,tPen\WObj:=wPaper;
    MoveL Offs(pOrigin,207.29,324.81,0.00),v60,z0,tPen\WObj:=wPaper;
    MoveL Offs(pOrigin,206.44,324.81,0.00),v40,z0,tPen\WObj:=wPaper;
    MoveL Offs(pOrigin,206.23,323.75,0.00),v40,fine,tPen\WObj:=wPaper;
    MoveL Offs(pOrigin,206.23,323.75,6.00),v60,z5,tPen\WObj:=wPaper;
    MoveL Offs(pOrigin,206.23,321.84,6.00),vTravel,z5,tPen\WObj:=wPaper;
    MoveL Offs(pOrigin,206.23,321.84,0.00),v60,z0,tPen\WObj:=wPaper;
    MoveL Offs(pOrigin,205.45,321.41,0.00),v40,z0,tPen\WObj:=wPaper;
    MoveL Offs(pOrigin,206.65,320.56,0.00),v40,z0,tPen\WObj:=wPaper;
    MoveL Offs(pOrigin,209.34,320.35,0.00),v40,z0,tPen\WObj:=wPaper;
    MoveL Offs(pOrigin,208.56,321.41,0.00),v40,z0,tPen\WObj:=wPaper;
    MoveL Offs(pOrigin,206.23,321.84,0.00),v40,fine,tPen\WObj:=wPaper;
    MoveL Offs(pOrigin,206.23,321.84,6.00),v60,z5,tPen\WObj:=wPaper;
    MoveL Offs(pOrigin,205.38,320.99,6.00),vTravel,z5,tPen\WObj:=wPaper;
    MoveL Offs(pOrigin,205.38,320.99,0.00),v60,z0,tPen\WObj:=wPaper;
    MoveL Offs(pOrigin,204.10,320.85,0.00),v40,z0,tPen\WObj:=wPaper;
    MoveL Offs(pOrigin,203.46,320.21,0.00),v40,z0,tPen\WObj:=wPaper;
    MoveL Offs(pOrigin,200.63,318.65,0.00),v40,z0,tPen\WObj:=wPaper;
    MoveL Offs(pOrigin,200.49,317.80,0.00),v40,z0,tPen\WObj:=wPaper;
    MoveL Offs(pOrigin,200.49,317.80,0.00),v40,z0,tPen\WObj:=wPaper;
    MoveL Offs(pOrigin,201.76,318.01,0.00),v40,z0,tPen\WObj:=wPaper;
    MoveL Offs(pOrigin,201.76,318.01,0.00),v40,z0,tPen\WObj:=wPaper;
    MoveL Offs(pOrigin,202.40,319.08,0.00),v40,z0,tPen\WObj:=wPaper;
    MoveL Offs(pOrigin,202.40,319.50,0.00),v40,z0,tPen\WObj:=wPaper;
    MoveL Offs(pOrigin,203.04,319.08,0.00),v40,z0,tPen\WObj:=wPaper;
    MoveL Offs(pOrigin,206.01,320.00,0.00),v40,z0,tPen\WObj:=wPaper;
    MoveL Offs(pOrigin,206.44,320.56,0.00),v40,fine,tPen\WObj:=wPaper;
    MoveL Offs(pOrigin,206.44,320.56,6.00),v60,z5,tPen\WObj:=wPaper;
    MoveL Offs(pOrigin,209.41,320.14,6.00),vTravel,z5,tPen\WObj:=wPaper;
    MoveL Offs(pOrigin,209.41,320.14,0.00),v60,z0,tPen\WObj:=wPaper;
    MoveL Offs(pOrigin,210.90,319.71,0.00),v40,z0,tPen\WObj:=wPaper;
    MoveL Offs(pOrigin,211.32,319.08,0.00),v40,z0,tPen\WObj:=wPaper;
    MoveL Offs(pOrigin,211.54,318.65,0.00),v40,z0,tPen\WObj:=wPaper;
    MoveL Offs(pOrigin,211.32,319.08,0.00),v40,fine,tPen\WObj:=wPaper;
    MoveL Offs(pOrigin,211.32,319.08,6.00),v60,z5,tPen\WObj:=wPaper;
    MoveL Offs(pOrigin,211.75,320.56,6.00),vTravel,z5,tPen\WObj:=wPaper;
    MoveL Offs(pOrigin,211.75,320.56,0.00),v60,z0,tPen\WObj:=wPaper;
    MoveL Offs(pOrigin,211.96,320.99,0.00),v40,z0,tPen\WObj:=wPaper;
    MoveL Offs(pOrigin,211.75,320.56,0.00),v40,fine,tPen\WObj:=wPaper;
    MoveL Offs(pOrigin,211.75,320.56,6.00),v60,z5,tPen\WObj:=wPaper;
    MoveL Offs(pOrigin,215.15,317.80,6.00),vTravel,z5,tPen\WObj:=wPaper;
    MoveL Offs(pOrigin,215.15,317.80,0.00),v60,z0,tPen\WObj:=wPaper;
    MoveL Offs(pOrigin,215.72,317.38,0.00),v40,z0,tPen\WObj:=wPaper;
    MoveL Offs(pOrigin,216.00,316.10,0.00),v40,z0,tPen\WObj:=wPaper;
    MoveL Offs(pOrigin,216.64,315.67,0.00),v40,fine,tPen\WObj:=wPaper;
    MoveL Offs(pOrigin,216.64,315.67,6.00),v60,z5,tPen\WObj:=wPaper;
    MoveL Offs(pOrigin,216.64,313.98,6.00),vTravel,z5,tPen\WObj:=wPaper;
    MoveL Offs(pOrigin,216.64,313.98,0.00),v60,z0,tPen\WObj:=wPaper;
    MoveL Offs(pOrigin,215.57,313.55,0.00),v40,z0,tPen\WObj:=wPaper;
    MoveL Offs(pOrigin,215.57,313.55,0.00),v40,z0,tPen\WObj:=wPaper;
    MoveL Offs(pOrigin,215.15,313.98,0.00),v40,z0,tPen\WObj:=wPaper;
    MoveL Offs(pOrigin,215.15,314.61,0.00),v40,z0,tPen\WObj:=wPaper;
    MoveL Offs(pOrigin,215.57,313.55,0.00),v40,z0,tPen\WObj:=wPaper;
    MoveL Offs(pOrigin,216.00,312.06,0.00),v40,z0,tPen\WObj:=wPaper;
    MoveL Offs(pOrigin,216.64,311.64,0.00),v40,z0,tPen\WObj:=wPaper;
    MoveL Offs(pOrigin,216.85,311.57,0.00),v40,z0,tPen\WObj:=wPaper;
    MoveL Offs(pOrigin,217.06,310.36,0.00),v40,z0,tPen\WObj:=wPaper;
    MoveL Offs(pOrigin,218.05,310.01,0.00),v40,z0,tPen\WObj:=wPaper;
    MoveL Offs(pOrigin,218.05,311.35,0.00),v40,z0,tPen\WObj:=wPaper;
    MoveL Offs(pOrigin,216.85,311.57,0.00),v40,z0,tPen\WObj:=wPaper;
    MoveL Offs(pOrigin,216.21,312.06,0.00),v40,z0,tPen\WObj:=wPaper;
    MoveL Offs(pOrigin,216.64,311.64,0.00),v40,z0,tPen\WObj:=wPaper;
    MoveL Offs(pOrigin,216.21,312.06,0.00),v40,fine,tPen\WObj:=wPaper;
    MoveL Offs(pOrigin,216.21,312.06,6.00),v60,z5,tPen\WObj:=wPaper;
    MoveL Offs(pOrigin,214.73,309.30,6.00),vTravel,z5,tPen\WObj:=wPaper;
    MoveL Offs(pOrigin,214.73,309.30,0.00),v60,z0,tPen\WObj:=wPaper;
    MoveL Offs(pOrigin,214.51,309.94,0.00),v40,z0,tPen\WObj:=wPaper;
    MoveL Offs(pOrigin,213.66,310.36,0.00),v40,z0,tPen\WObj:=wPaper;
    MoveL Offs(pOrigin,213.24,311.00,0.00),v40,fine,tPen\WObj:=wPaper;
    MoveL Offs(pOrigin,213.24,311.00,6.00),v60,z5,tPen\WObj:=wPaper;
    MoveL Offs(pOrigin,211.75,311.42,6.00),vTravel,z5,tPen\WObj:=wPaper;
    MoveL Offs(pOrigin,211.75,311.42,0.00),v60,z0,tPen\WObj:=wPaper;
    MoveL Offs(pOrigin,210.69,311.42,0.00),v40,z0,tPen\WObj:=wPaper;
    MoveL Offs(pOrigin,210.05,312.06,0.00),v40,z0,tPen\WObj:=wPaper;
    MoveL Offs(pOrigin,210.26,311.85,0.00),v40,z0,tPen\WObj:=wPaper;
    MoveL Offs(pOrigin,209.84,312.06,0.00),v40,z0,tPen\WObj:=wPaper;
    MoveL Offs(pOrigin,207.93,313.41,0.00),v40,z0,tPen\WObj:=wPaper;
    MoveL Offs(pOrigin,206.65,313.55,0.00),v40,fine,tPen\WObj:=wPaper;
    MoveL Offs(pOrigin,206.65,313.55,6.00),v60,z5,tPen\WObj:=wPaper;
    MoveL Offs(pOrigin,205.16,314.40,6.00),vTravel,z5,tPen\WObj:=wPaper;
    MoveL Offs(pOrigin,205.16,314.40,0.00),v60,z0,tPen\WObj:=wPaper;
    MoveL Offs(pOrigin,204.74,315.04,0.00),v40,z0,tPen\WObj:=wPaper;
    MoveL Offs(pOrigin,203.89,315.04,0.00),v40,z0,tPen\WObj:=wPaper;
    MoveL Offs(pOrigin,203.89,315.04,0.00),v40,z0,tPen\WObj:=wPaper;
    MoveL Offs(pOrigin,203.25,315.25,0.00),v40,z0,tPen\WObj:=wPaper;
    MoveL Offs(pOrigin,203.04,315.67,0.00),v40,z0,tPen\WObj:=wPaper;
    MoveL Offs(pOrigin,203.04,315.67,0.00),v40,z0,tPen\WObj:=wPaper;
    MoveL Offs(pOrigin,200.06,314.54,0.00),v40,z0,tPen\WObj:=wPaper;
    MoveL Offs(pOrigin,199.43,313.83,0.00),v40,z0,tPen\WObj:=wPaper;
    MoveL Offs(pOrigin,197.30,312.70,0.00),v40,z0,tPen\WObj:=wPaper;
    MoveL Offs(pOrigin,196.88,311.64,0.00),v40,z0,tPen\WObj:=wPaper;
    MoveL Offs(pOrigin,196.88,311.64,0.00),v40,z0,tPen\WObj:=wPaper;
    MoveL Offs(pOrigin,200.49,312.49,0.00),v40,z0,tPen\WObj:=wPaper;
    MoveL Offs(pOrigin,203.46,312.49,0.00),v40,z0,tPen\WObj:=wPaper;
    MoveL Offs(pOrigin,206.44,311.57,0.00),v40,z0,tPen\WObj:=wPaper;
    MoveL Offs(pOrigin,206.86,310.58,0.00),v40,z0,tPen\WObj:=wPaper;
    MoveL Offs(pOrigin,206.86,310.58,0.00),v40,z0,tPen\WObj:=wPaper;
    MoveL Offs(pOrigin,206.65,310.01,0.00),v40,z0,tPen\WObj:=wPaper;
    MoveL Offs(pOrigin,205.80,309.94,0.00),v40,z0,tPen\WObj:=wPaper;
    MoveL Offs(pOrigin,203.46,311.42,0.00),v40,z0,tPen\WObj:=wPaper;
    MoveL Offs(pOrigin,200.91,311.42,0.00),v40,z0,tPen\WObj:=wPaper;
    MoveL Offs(pOrigin,198.15,310.43,0.00),v40,z0,tPen\WObj:=wPaper;
    MoveL Offs(pOrigin,194.75,307.17,0.00),v40,z0,tPen\WObj:=wPaper;
    MoveL Offs(pOrigin,193.55,305.48,0.00),v40,z0,tPen\WObj:=wPaper;
    MoveL Offs(pOrigin,193.26,304.62,0.00),v40,z0,tPen\WObj:=wPaper;
    MoveL Offs(pOrigin,193.90,303.99,0.00),v40,fine,tPen\WObj:=wPaper;
    MoveL Offs(pOrigin,193.90,303.99,6.00),v60,z5,tPen\WObj:=wPaper;
    MoveL Offs(pOrigin,194.11,306.11,6.00),vTravel,z5,tPen\WObj:=wPaper;
  ENDPROC

  PROC DrawPart40()
    MoveL Offs(pOrigin,194.11,306.11,0.00),v60,z0,tPen\WObj:=wPaper;
    MoveL Offs(pOrigin,194.54,306.54,0.00),v40,z0,tPen\WObj:=wPaper;
    MoveL Offs(pOrigin,194.11,306.11,0.00),v40,z0,tPen\WObj:=wPaper;
    MoveL Offs(pOrigin,194.75,306.96,0.00),v40,z0,tPen\WObj:=wPaper;
    MoveL Offs(pOrigin,195.60,307.81,0.00),v40,z0,tPen\WObj:=wPaper;
    MoveL Offs(pOrigin,194.75,306.96,0.00),v40,fine,tPen\WObj:=wPaper;
    MoveL Offs(pOrigin,194.75,306.96,6.00),v60,z5,tPen\WObj:=wPaper;
    MoveL Offs(pOrigin,194.32,308.66,6.00),vTravel,z5,tPen\WObj:=wPaper;
    MoveL Offs(pOrigin,194.32,308.66,0.00),v60,z0,tPen\WObj:=wPaper;
    MoveL Offs(pOrigin,195.60,310.58,0.00),v40,z0,tPen\WObj:=wPaper;
    MoveL Offs(pOrigin,196.88,311.64,0.00),v40,fine,tPen\WObj:=wPaper;
    MoveL Offs(pOrigin,196.88,311.64,6.00),v60,z5,tPen\WObj:=wPaper;
    MoveL Offs(pOrigin,196.02,314.61,6.00),vTravel,z5,tPen\WObj:=wPaper;
    MoveL Offs(pOrigin,196.02,314.61,0.00),v60,z0,tPen\WObj:=wPaper;
    MoveL Offs(pOrigin,197.09,315.67,0.00),v40,z0,tPen\WObj:=wPaper;
    MoveL Offs(pOrigin,197.09,315.67,0.00),v40,z0,tPen\WObj:=wPaper;
    MoveL Offs(pOrigin,197.02,316.31,0.00),v40,z0,tPen\WObj:=wPaper;
    MoveL Offs(pOrigin,197.73,317.38,0.00),v40,z0,tPen\WObj:=wPaper;
    MoveL Offs(pOrigin,202.61,321.41,0.00),v40,fine,tPen\WObj:=wPaper;
    MoveL Offs(pOrigin,202.61,321.41,6.00),v60,z5,tPen\WObj:=wPaper;
    MoveL Offs(pOrigin,200.70,320.14,6.00),vTravel,z5,tPen\WObj:=wPaper;
    MoveL Offs(pOrigin,200.70,320.14,0.00),v60,z0,tPen\WObj:=wPaper;
    MoveL Offs(pOrigin,201.12,320.35,0.00),v40,z0,tPen\WObj:=wPaper;
    MoveL Offs(pOrigin,200.70,320.14,0.00),v40,fine,tPen\WObj:=wPaper;
    MoveL Offs(pOrigin,200.70,320.14,6.00),v60,z5,tPen\WObj:=wPaper;
    MoveL Offs(pOrigin,199.43,319.08,6.00),vTravel,z5,tPen\WObj:=wPaper;
    MoveL Offs(pOrigin,199.43,319.08,0.00),v60,z0,tPen\WObj:=wPaper;
    MoveL Offs(pOrigin,200.06,319.71,0.00),v40,z0,tPen\WObj:=wPaper;
    MoveL Offs(pOrigin,199.43,319.08,0.00),v40,fine,tPen\WObj:=wPaper;
    MoveL Offs(pOrigin,199.43,319.08,6.00),v60,z5,tPen\WObj:=wPaper;
    MoveL Offs(pOrigin,198.36,318.23,6.00),vTravel,z5,tPen\WObj:=wPaper;
    MoveL Offs(pOrigin,198.36,318.23,0.00),v60,z0,tPen\WObj:=wPaper;
    MoveL Offs(pOrigin,199.21,318.86,0.00),v40,z0,tPen\WObj:=wPaper;
    MoveL Offs(pOrigin,198.36,318.23,0.00),v40,z0,tPen\WObj:=wPaper;
    MoveL Offs(pOrigin,197.73,317.59,0.00),v40,z0,tPen\WObj:=wPaper;
    MoveL Offs(pOrigin,198.15,318.01,0.00),v40,z0,tPen\WObj:=wPaper;
    MoveL Offs(pOrigin,197.73,317.59,0.00),v40,fine,tPen\WObj:=wPaper;
    MoveL Offs(pOrigin,197.73,317.59,6.00),v60,z5,tPen\WObj:=wPaper;
    MoveL Offs(pOrigin,197.09,318.65,6.00),vTravel,z5,tPen\WObj:=wPaper;
    MoveL Offs(pOrigin,197.09,318.65,0.00),v60,z0,tPen\WObj:=wPaper;
    MoveL Offs(pOrigin,197.51,319.08,0.00),v40,z0,tPen\WObj:=wPaper;
    MoveL Offs(pOrigin,197.09,318.65,0.00),v40,z0,tPen\WObj:=wPaper;
    MoveL Offs(pOrigin,197.73,319.50,0.00),v40,z0,tPen\WObj:=wPaper;
    MoveL Offs(pOrigin,198.15,319.92,0.00),v40,z0,tPen\WObj:=wPaper;
    MoveL Offs(pOrigin,197.73,319.50,0.00),v40,fine,tPen\WObj:=wPaper;
    MoveL Offs(pOrigin,197.73,319.50,6.00),v60,z5,tPen\WObj:=wPaper;
    MoveL Offs(pOrigin,196.45,317.59,6.00),vTravel,z5,tPen\WObj:=wPaper;
    MoveL Offs(pOrigin,196.45,317.59,0.00),v60,z0,tPen\WObj:=wPaper;
    MoveL Offs(pOrigin,196.66,318.01,0.00),v40,z0,tPen\WObj:=wPaper;
    MoveL Offs(pOrigin,196.45,317.59,0.00),v40,fine,tPen\WObj:=wPaper;
    MoveL Offs(pOrigin,196.45,317.59,6.00),v60,z5,tPen\WObj:=wPaper;
    MoveL Offs(pOrigin,197.09,315.67,6.00),vTravel,z5,tPen\WObj:=wPaper;
    MoveL Offs(pOrigin,197.09,315.67,0.00),v60,z0,tPen\WObj:=wPaper;
    MoveL Offs(pOrigin,198.15,316.10,0.00),v40,z0,tPen\WObj:=wPaper;
    MoveL Offs(pOrigin,199.64,317.52,0.00),v40,z0,tPen\WObj:=wPaper;
    MoveL Offs(pOrigin,200.49,317.80,0.00),v40,fine,tPen\WObj:=wPaper;
    MoveL Offs(pOrigin,200.49,317.80,6.00),v60,z5,tPen\WObj:=wPaper;
    MoveL Offs(pOrigin,201.76,318.01,6.00),vTravel,z5,tPen\WObj:=wPaper;
    MoveL Offs(pOrigin,201.76,318.01,0.00),v60,z0,tPen\WObj:=wPaper;
    MoveL Offs(pOrigin,202.19,317.80,0.00),v40,z0,tPen\WObj:=wPaper;
    MoveL Offs(pOrigin,205.59,318.23,0.00),v40,z0,tPen\WObj:=wPaper;
    MoveL Offs(pOrigin,207.50,318.01,0.00),v40,z0,tPen\WObj:=wPaper;
    MoveL Offs(pOrigin,208.92,317.52,0.00),v40,z0,tPen\WObj:=wPaper;
    MoveL Offs(pOrigin,209.20,316.95,0.00),v40,fine,tPen\WObj:=wPaper;
    MoveL Offs(pOrigin,209.20,316.95,6.00),v60,z5,tPen\WObj:=wPaper;
    MoveL Offs(pOrigin,211.32,315.67,6.00),vTravel,z5,tPen\WObj:=wPaper;
    MoveL Offs(pOrigin,211.32,315.67,0.00),v60,z0,tPen\WObj:=wPaper;
    MoveL Offs(pOrigin,211.40,314.61,0.00),v40,z0,tPen\WObj:=wPaper;
    MoveL Offs(pOrigin,212.39,313.34,0.00),v40,z0,tPen\WObj:=wPaper;
    MoveL Offs(pOrigin,213.02,313.12,0.00),v40,z0,tPen\WObj:=wPaper;
    MoveL Offs(pOrigin,213.02,313.12,0.00),v40,z0,tPen\WObj:=wPaper;
    MoveL Offs(pOrigin,213.45,311.64,0.00),v40,z0,tPen\WObj:=wPaper;
    MoveL Offs(pOrigin,213.24,311.21,0.00),v40,z0,tPen\WObj:=wPaper;
    MoveL Offs(pOrigin,212.60,311.00,0.00),v40,z0,tPen\WObj:=wPaper;
    MoveL Offs(pOrigin,211.75,311.64,0.00),v40,z0,tPen\WObj:=wPaper;
    MoveL Offs(pOrigin,211.32,312.70,0.00),v40,z0,tPen\WObj:=wPaper;
    MoveL Offs(pOrigin,208.99,314.83,0.00),v40,z0,tPen\WObj:=wPaper;
    MoveL Offs(pOrigin,205.38,316.10,0.00),v40,fine,tPen\WObj:=wPaper;
    MoveL Offs(pOrigin,205.38,316.10,6.00),v60,z5,tPen\WObj:=wPaper;
    MoveL Offs(pOrigin,209.20,314.40,6.00),vTravel,z5,tPen\WObj:=wPaper;
    MoveL Offs(pOrigin,209.20,314.40,0.00),v60,z0,tPen\WObj:=wPaper;
    MoveL Offs(pOrigin,208.77,314.83,0.00),v40,z0,tPen\WObj:=wPaper;
    MoveL Offs(pOrigin,209.20,314.40,0.00),v40,z0,tPen\WObj:=wPaper;
    MoveL Offs(pOrigin,210.05,313.76,0.00),v40,z0,tPen\WObj:=wPaper;
    MoveL Offs(pOrigin,209.62,314.19,0.00),v40,z0,tPen\WObj:=wPaper;
    MoveL Offs(pOrigin,210.05,313.76,0.00),v40,fine,tPen\WObj:=wPaper;
    MoveL Offs(pOrigin,210.05,313.76,6.00),v60,z5,tPen\WObj:=wPaper;
    MoveL Offs(pOrigin,210.90,312.91,6.00),vTravel,z5,tPen\WObj:=wPaper;
    MoveL Offs(pOrigin,210.90,312.91,0.00),v60,z0,tPen\WObj:=wPaper;
    MoveL Offs(pOrigin,210.26,313.55,0.00),v40,z0,tPen\WObj:=wPaper;
    MoveL Offs(pOrigin,210.90,312.91,0.00),v40,fine,tPen\WObj:=wPaper;
    MoveL Offs(pOrigin,210.90,312.91,6.00),v60,z5,tPen\WObj:=wPaper;
    MoveL Offs(pOrigin,213.02,313.12,6.00),vTravel,z5,tPen\WObj:=wPaper;
    MoveL Offs(pOrigin,213.02,313.12,0.00),v60,z0,tPen\WObj:=wPaper;
    MoveL Offs(pOrigin,213.24,313.55,0.00),v40,z0,tPen\WObj:=wPaper;
    MoveL Offs(pOrigin,212.88,314.61,0.00),v40,z0,tPen\WObj:=wPaper;
    MoveL Offs(pOrigin,211.96,315.67,0.00),v40,fine,tPen\WObj:=wPaper;
    MoveL Offs(pOrigin,211.96,315.67,6.00),v60,z5,tPen\WObj:=wPaper;
    MoveL Offs(pOrigin,212.81,314.40,6.00),vTravel,z5,tPen\WObj:=wPaper;
    MoveL Offs(pOrigin,212.81,314.40,0.00),v60,z0,tPen\WObj:=wPaper;
    MoveL Offs(pOrigin,212.60,314.83,0.00),v40,z0,tPen\WObj:=wPaper;
    MoveL Offs(pOrigin,212.81,314.40,0.00),v40,fine,tPen\WObj:=wPaper;
    MoveL Offs(pOrigin,212.81,314.40,6.00),v60,z5,tPen\WObj:=wPaper;
    MoveL Offs(pOrigin,210.26,309.94,6.00),vTravel,z5,tPen\WObj:=wPaper;
    MoveL Offs(pOrigin,210.26,309.94,0.00),v60,z0,tPen\WObj:=wPaper;
    MoveL Offs(pOrigin,209.20,309.94,0.00),v40,z0,tPen\WObj:=wPaper;
    MoveL Offs(pOrigin,208.56,310.58,0.00),v40,z0,tPen\WObj:=wPaper;
    MoveL Offs(pOrigin,208.77,310.36,0.00),v40,z0,tPen\WObj:=wPaper;
    MoveL Offs(pOrigin,208.35,310.58,0.00),v40,z0,tPen\WObj:=wPaper;
    MoveL Offs(pOrigin,207.29,310.79,0.00),v40,z0,tPen\WObj:=wPaper;
    MoveL Offs(pOrigin,206.86,310.58,0.00),v40,z0,tPen\WObj:=wPaper;
    MoveL Offs(pOrigin,206.86,309.94,0.00),v40,z0,tPen\WObj:=wPaper;
    MoveL Offs(pOrigin,207.50,309.23,0.00),v40,z0,tPen\WObj:=wPaper;
    MoveL Offs(pOrigin,209.84,308.02,0.00),v40,fine,tPen\WObj:=wPaper;
    MoveL Offs(pOrigin,209.84,308.02,6.00),v60,z5,tPen\WObj:=wPaper;
    MoveL Offs(pOrigin,210.69,306.96,6.00),vTravel,z5,tPen\WObj:=wPaper;
    MoveL Offs(pOrigin,210.69,306.96,0.00),v60,z0,tPen\WObj:=wPaper;
    MoveL Offs(pOrigin,211.96,306.75,0.00),v40,z0,tPen\WObj:=wPaper;
    MoveL Offs(pOrigin,212.81,305.97,0.00),v40,z0,tPen\WObj:=wPaper;
    MoveL Offs(pOrigin,213.88,305.69,0.00),v40,z0,tPen\WObj:=wPaper;
  ENDPROC

  PROC DrawPart41()
    MoveL Offs(pOrigin,213.88,305.69,0.00),v40,z0,tPen\WObj:=wPaper;
    MoveL Offs(pOrigin,213.80,303.77,0.00),v40,z0,tPen\WObj:=wPaper;
    MoveL Offs(pOrigin,212.81,303.35,0.00),v40,z0,tPen\WObj:=wPaper;
    MoveL Offs(pOrigin,211.96,303.56,0.00),v40,z0,tPen\WObj:=wPaper;
    MoveL Offs(pOrigin,211.96,303.56,0.00),v40,z0,tPen\WObj:=wPaper;
    MoveL Offs(pOrigin,213.45,305.69,0.00),v40,z0,tPen\WObj:=wPaper;
    MoveL Offs(pOrigin,212.60,305.90,0.00),v40,z0,tPen\WObj:=wPaper;
    MoveL Offs(pOrigin,211.32,305.26,0.00),v40,z0,tPen\WObj:=wPaper;
    MoveL Offs(pOrigin,208.14,304.77,0.00),v40,z0,tPen\WObj:=wPaper;
    MoveL Offs(pOrigin,206.86,303.77,0.00),v40,z0,tPen\WObj:=wPaper;
    MoveL Offs(pOrigin,206.86,303.77,0.00),v40,z0,tPen\WObj:=wPaper;
    MoveL Offs(pOrigin,206.01,303.99,0.00),v40,z0,tPen\WObj:=wPaper;
    MoveL Offs(pOrigin,205.38,303.00,0.00),v40,z0,tPen\WObj:=wPaper;
    MoveL Offs(pOrigin,201.34,301.86,0.00),v40,z0,tPen\WObj:=wPaper;
    MoveL Offs(pOrigin,201.34,302.92,0.00),v40,z0,tPen\WObj:=wPaper;
    MoveL Offs(pOrigin,200.70,303.14,0.00),v40,z0,tPen\WObj:=wPaper;
    MoveL Offs(pOrigin,198.79,302.36,0.00),v40,z0,tPen\WObj:=wPaper;
    MoveL Offs(pOrigin,198.36,302.50,0.00),v40,z0,tPen\WObj:=wPaper;
    MoveL Offs(pOrigin,198.36,302.29,0.00),v40,z0,tPen\WObj:=wPaper;
    MoveL Offs(pOrigin,195.88,298.67,0.00),v40,z0,tPen\WObj:=wPaper;
    MoveL Offs(pOrigin,194.96,295.06,0.00),v40,z0,tPen\WObj:=wPaper;
    MoveL Offs(pOrigin,194.96,295.06,0.00),v40,z0,tPen\WObj:=wPaper;
    MoveL Offs(pOrigin,196.45,295.49,0.00),v40,z0,tPen\WObj:=wPaper;
    MoveL Offs(pOrigin,196.45,295.49,0.00),v40,z0,tPen\WObj:=wPaper;
    MoveL Offs(pOrigin,197.51,297.19,0.00),v40,z0,tPen\WObj:=wPaper;
    MoveL Offs(pOrigin,199.64,299.31,0.00),v40,fine,tPen\WObj:=wPaper;
    MoveL Offs(pOrigin,199.64,299.31,6.00),v60,z5,tPen\WObj:=wPaper;
    MoveL Offs(pOrigin,199.64,300.59,6.00),vTravel,z5,tPen\WObj:=wPaper;
    MoveL Offs(pOrigin,199.64,300.59,0.00),v60,z0,tPen\WObj:=wPaper;
    MoveL Offs(pOrigin,200.06,300.80,0.00),v40,z0,tPen\WObj:=wPaper;
    MoveL Offs(pOrigin,199.64,300.59,0.00),v40,fine,tPen\WObj:=wPaper;
    MoveL Offs(pOrigin,199.64,300.59,6.00),v60,z5,tPen\WObj:=wPaper;
    MoveL Offs(pOrigin,197.30,300.38,6.00),vTravel,z5,tPen\WObj:=wPaper;
    MoveL Offs(pOrigin,197.30,300.38,0.00),v60,z0,tPen\WObj:=wPaper;
    MoveL Offs(pOrigin,197.94,301.23,0.00),v40,z0,tPen\WObj:=wPaper;
    MoveL Offs(pOrigin,197.30,300.38,0.00),v40,fine,tPen\WObj:=wPaper;
    MoveL Offs(pOrigin,197.30,300.38,6.00),v60,z5,tPen\WObj:=wPaper;
    MoveL Offs(pOrigin,195.60,300.16,6.00),vTravel,z5,tPen\WObj:=wPaper;
    MoveL Offs(pOrigin,195.60,300.16,0.00),v60,z0,tPen\WObj:=wPaper;
    MoveL Offs(pOrigin,196.02,300.80,0.00),v40,z0,tPen\WObj:=wPaper;
    MoveL Offs(pOrigin,195.60,300.16,0.00),v40,z0,tPen\WObj:=wPaper;
    MoveL Offs(pOrigin,195.18,299.52,0.00),v40,z0,tPen\WObj:=wPaper;
    MoveL Offs(pOrigin,195.39,299.95,0.00),v40,z0,tPen\WObj:=wPaper;
    MoveL Offs(pOrigin,195.18,299.52,0.00),v40,fine,tPen\WObj:=wPaper;
    MoveL Offs(pOrigin,195.18,299.52,6.00),v60,z5,tPen\WObj:=wPaper;
    MoveL Offs(pOrigin,196.45,295.49,6.00),vTravel,z5,tPen\WObj:=wPaper;
    MoveL Offs(pOrigin,196.45,295.49,0.00),v60,z0,tPen\WObj:=wPaper;
    MoveL Offs(pOrigin,196.31,294.42,0.00),v40,z0,tPen\WObj:=wPaper;
    MoveL Offs(pOrigin,194.11,289.96,0.00),v40,z0,tPen\WObj:=wPaper;
    MoveL Offs(pOrigin,193.90,289.54,0.00),v40,z0,tPen\WObj:=wPaper;
    MoveL Offs(pOrigin,194.11,289.96,0.00),v40,z0,tPen\WObj:=wPaper;
    MoveL Offs(pOrigin,193.90,289.54,0.00),v40,fine,tPen\WObj:=wPaper;
    MoveL Offs(pOrigin,193.90,289.54,6.00),v60,z5,tPen\WObj:=wPaper;
    MoveL Offs(pOrigin,193.90,287.20,6.00),vTravel,z5,tPen\WObj:=wPaper;
    MoveL Offs(pOrigin,193.90,287.20,0.00),v60,z0,tPen\WObj:=wPaper;
    MoveL Offs(pOrigin,193.69,286.14,0.00),v40,z0,tPen\WObj:=wPaper;
    MoveL Offs(pOrigin,193.69,286.14,0.00),v40,z0,tPen\WObj:=wPaper;
    MoveL Offs(pOrigin,193.90,285.50,0.00),v40,z0,tPen\WObj:=wPaper;
    MoveL Offs(pOrigin,192.98,284.01,0.00),v40,z0,tPen\WObj:=wPaper;
    MoveL Offs(pOrigin,192.84,282.52,0.00),v40,fine,tPen\WObj:=wPaper;
    MoveL Offs(pOrigin,192.84,282.52,6.00),v60,z5,tPen\WObj:=wPaper;
    MoveL Offs(pOrigin,193.05,284.44,6.00),vTravel,z5,tPen\WObj:=wPaper;
    MoveL Offs(pOrigin,193.05,284.44,0.00),v60,z0,tPen\WObj:=wPaper;
    MoveL Offs(pOrigin,192.84,285.29,0.00),v40,z0,tPen\WObj:=wPaper;
    MoveL Offs(pOrigin,193.69,286.14,0.00),v40,z0,tPen\WObj:=wPaper;
    MoveL Offs(pOrigin,193.90,287.20,0.00),v40,z0,tPen\WObj:=wPaper;
    MoveL Offs(pOrigin,194.96,287.62,0.00),v40,z0,tPen\WObj:=wPaper;
    MoveL Offs(pOrigin,196.17,290.17,0.00),v40,z0,tPen\WObj:=wPaper;
    MoveL Offs(pOrigin,198.36,293.58,0.00),v40,z0,tPen\WObj:=wPaper;
    MoveL Offs(pOrigin,199.64,294.71,0.00),v40,z0,tPen\WObj:=wPaper;
    MoveL Offs(pOrigin,201.12,294.64,0.00),v40,z0,tPen\WObj:=wPaper;
    MoveL Offs(pOrigin,201.12,293.79,0.00),v40,z0,tPen\WObj:=wPaper;
    MoveL Offs(pOrigin,201.05,293.15,0.00),v40,z0,tPen\WObj:=wPaper;
    MoveL Offs(pOrigin,200.20,291.88,0.00),v40,z0,tPen\WObj:=wPaper;
    MoveL Offs(pOrigin,199.43,291.45,0.00),v40,z0,tPen\WObj:=wPaper;
    MoveL Offs(pOrigin,200.27,291.66,0.00),v40,z0,tPen\WObj:=wPaper;
    MoveL Offs(pOrigin,200.70,291.02,0.00),v40,z0,tPen\WObj:=wPaper;
    MoveL Offs(pOrigin,200.13,289.54,0.00),v40,z0,tPen\WObj:=wPaper;
    MoveL Offs(pOrigin,198.15,286.56,0.00),v40,z0,tPen\WObj:=wPaper;
    MoveL Offs(pOrigin,197.30,286.14,0.00),v40,z0,tPen\WObj:=wPaper;
    MoveL Offs(pOrigin,198.36,286.56,0.00),v40,z0,tPen\WObj:=wPaper;
    MoveL Offs(pOrigin,198.79,287.20,0.00),v40,z0,tPen\WObj:=wPaper;
    MoveL Offs(pOrigin,198.36,286.56,0.00),v40,z0,tPen\WObj:=wPaper;
    MoveL Offs(pOrigin,197.73,287.41,0.00),v40,z0,tPen\WObj:=wPaper;
    MoveL Offs(pOrigin,197.94,287.84,0.00),v40,z0,tPen\WObj:=wPaper;
    MoveL Offs(pOrigin,197.73,287.41,0.00),v40,fine,tPen\WObj:=wPaper;
    MoveL Offs(pOrigin,197.73,287.41,6.00),v60,z5,tPen\WObj:=wPaper;
    MoveL Offs(pOrigin,196.66,288.05,6.00),vTravel,z5,tPen\WObj:=wPaper;
    MoveL Offs(pOrigin,196.66,288.05,0.00),v60,z0,tPen\WObj:=wPaper;
    MoveL Offs(pOrigin,196.88,288.48,0.00),v40,z0,tPen\WObj:=wPaper;
    MoveL Offs(pOrigin,196.66,288.05,0.00),v40,z0,tPen\WObj:=wPaper;
    MoveL Offs(pOrigin,197.09,288.90,0.00),v40,z0,tPen\WObj:=wPaper;
    MoveL Offs(pOrigin,197.30,289.33,0.00),v40,z0,tPen\WObj:=wPaper;
    MoveL Offs(pOrigin,197.09,288.90,0.00),v40,fine,tPen\WObj:=wPaper;
    MoveL Offs(pOrigin,197.09,288.90,6.00),v60,z5,tPen\WObj:=wPaper;
    MoveL Offs(pOrigin,198.57,288.90,6.00),vTravel,z5,tPen\WObj:=wPaper;
    MoveL Offs(pOrigin,198.57,288.90,0.00),v60,z0,tPen\WObj:=wPaper;
    MoveL Offs(pOrigin,198.79,289.33,0.00),v40,z0,tPen\WObj:=wPaper;
    MoveL Offs(pOrigin,198.57,288.90,0.00),v40,fine,tPen\WObj:=wPaper;
    MoveL Offs(pOrigin,198.57,288.90,6.00),v60,z5,tPen\WObj:=wPaper;
    MoveL Offs(pOrigin,197.94,290.39,6.00),vTravel,z5,tPen\WObj:=wPaper;
    MoveL Offs(pOrigin,197.94,290.39,0.00),v60,z0,tPen\WObj:=wPaper;
    MoveL Offs(pOrigin,198.15,290.81,0.00),v40,z0,tPen\WObj:=wPaper;
    MoveL Offs(pOrigin,197.94,290.39,0.00),v40,fine,tPen\WObj:=wPaper;
    MoveL Offs(pOrigin,197.94,290.39,6.00),v60,z5,tPen\WObj:=wPaper;
    MoveL Offs(pOrigin,195.81,291.66,6.00),vTravel,z5,tPen\WObj:=wPaper;
    MoveL Offs(pOrigin,195.81,291.66,0.00),v60,z0,tPen\WObj:=wPaper;
    MoveL Offs(pOrigin,196.24,292.30,0.00),v40,z0,tPen\WObj:=wPaper;
    MoveL Offs(pOrigin,195.81,291.66,0.00),v40,fine,tPen\WObj:=wPaper;
    MoveL Offs(pOrigin,195.81,291.66,6.00),v60,z5,tPen\WObj:=wPaper;
    MoveL Offs(pOrigin,195.18,292.73,6.00),vTravel,z5,tPen\WObj:=wPaper;
    MoveL Offs(pOrigin,195.18,292.73,0.00),v60,z0,tPen\WObj:=wPaper;
    MoveL Offs(pOrigin,195.60,293.36,0.00),v40,z0,tPen\WObj:=wPaper;
    MoveL Offs(pOrigin,195.18,292.73,0.00),v40,fine,tPen\WObj:=wPaper;
    MoveL Offs(pOrigin,195.18,292.73,6.00),v60,z5,tPen\WObj:=wPaper;
    MoveL Offs(pOrigin,193.26,291.88,6.00),vTravel,z5,tPen\WObj:=wPaper;
    MoveL Offs(pOrigin,193.26,291.88,0.00),v60,z0,tPen\WObj:=wPaper;
    MoveL Offs(pOrigin,194.96,295.06,0.00),v40,fine,tPen\WObj:=wPaper;
    MoveL Offs(pOrigin,194.96,295.06,6.00),v60,z5,tPen\WObj:=wPaper;
    MoveL Offs(pOrigin,197.73,294.42,6.00),vTravel,z5,tPen\WObj:=wPaper;
  ENDPROC

  PROC DrawPart42()
    MoveL Offs(pOrigin,197.73,294.42,0.00),v60,z0,tPen\WObj:=wPaper;
    MoveL Offs(pOrigin,198.15,294.85,0.00),v40,z0,tPen\WObj:=wPaper;
    MoveL Offs(pOrigin,197.73,294.42,0.00),v40,fine,tPen\WObj:=wPaper;
    MoveL Offs(pOrigin,197.73,294.42,6.00),v60,z5,tPen\WObj:=wPaper;
    MoveL Offs(pOrigin,198.79,295.49,6.00),vTravel,z5,tPen\WObj:=wPaper;
    MoveL Offs(pOrigin,198.79,295.49,0.00),v60,z0,tPen\WObj:=wPaper;
    MoveL Offs(pOrigin,199.21,296.12,0.00),v40,z0,tPen\WObj:=wPaper;
    MoveL Offs(pOrigin,198.79,295.49,0.00),v40,z0,tPen\WObj:=wPaper;
    MoveL Offs(pOrigin,199.43,296.34,0.00),v40,z0,tPen\WObj:=wPaper;
    MoveL Offs(pOrigin,200.27,297.19,0.00),v40,z0,tPen\WObj:=wPaper;
    MoveL Offs(pOrigin,199.43,296.34,0.00),v40,fine,tPen\WObj:=wPaper;
    MoveL Offs(pOrigin,199.43,296.34,6.00),v60,z5,tPen\WObj:=wPaper;
    MoveL Offs(pOrigin,202.40,299.95,6.00),vTravel,z5,tPen\WObj:=wPaper;
    MoveL Offs(pOrigin,202.40,299.95,0.00),v60,z0,tPen\WObj:=wPaper;
    MoveL Offs(pOrigin,204.95,301.01,0.00),v40,fine,tPen\WObj:=wPaper;
    MoveL Offs(pOrigin,204.95,301.01,6.00),v60,z5,tPen\WObj:=wPaper;
    MoveL Offs(pOrigin,205.59,302.92,6.00),vTravel,z5,tPen\WObj:=wPaper;
    MoveL Offs(pOrigin,205.59,302.92,0.00),v60,z0,tPen\WObj:=wPaper;
    MoveL Offs(pOrigin,206.65,303.14,0.00),v40,z0,tPen\WObj:=wPaper;
    MoveL Offs(pOrigin,206.86,303.77,0.00),v40,fine,tPen\WObj:=wPaper;
    MoveL Offs(pOrigin,206.86,303.77,6.00),v60,z5,tPen\WObj:=wPaper;
    MoveL Offs(pOrigin,207.71,302.29,6.00),vTravel,z5,tPen\WObj:=wPaper;
    MoveL Offs(pOrigin,207.71,302.29,0.00),v60,z0,tPen\WObj:=wPaper;
    MoveL Offs(pOrigin,211.96,303.56,0.00),v40,z0,tPen\WObj:=wPaper;
    MoveL Offs(pOrigin,211.96,303.35,0.00),v40,z0,tPen\WObj:=wPaper;
    MoveL Offs(pOrigin,211.47,301.86,0.00),v40,z0,tPen\WObj:=wPaper;
    MoveL Offs(pOrigin,209.84,301.01,0.00),v40,z0,tPen\WObj:=wPaper;
    MoveL Offs(pOrigin,209.84,301.01,0.00),v40,z0,tPen\WObj:=wPaper;
    MoveL Offs(pOrigin,207.93,300.66,0.00),v40,z0,tPen\WObj:=wPaper;
    MoveL Offs(pOrigin,207.29,300.02,0.00),v40,z0,tPen\WObj:=wPaper;
    MoveL Offs(pOrigin,205.80,300.23,0.00),v40,z0,tPen\WObj:=wPaper;
    MoveL Offs(pOrigin,202.82,298.53,0.00),v40,z0,tPen\WObj:=wPaper;
    MoveL Offs(pOrigin,202.40,298.89,0.00),v40,z0,tPen\WObj:=wPaper;
    MoveL Offs(pOrigin,202.40,299.95,0.00),v40,fine,tPen\WObj:=wPaper;
    MoveL Offs(pOrigin,202.40,299.95,6.00),v60,z5,tPen\WObj:=wPaper;
    MoveL Offs(pOrigin,204.74,296.98,6.00),vTravel,z5,tPen\WObj:=wPaper;
    MoveL Offs(pOrigin,204.74,296.98,0.00),v60,z0,tPen\WObj:=wPaper;
    MoveL Offs(pOrigin,204.52,296.55,0.00),v40,z0,tPen\WObj:=wPaper;
    MoveL Offs(pOrigin,204.95,296.12,0.00),v40,z0,tPen\WObj:=wPaper;
    MoveL Offs(pOrigin,207.50,296.76,0.00),v40,z0,tPen\WObj:=wPaper;
    MoveL Offs(pOrigin,207.50,296.76,0.00),v40,z0,tPen\WObj:=wPaper;
    MoveL Offs(pOrigin,207.29,295.06,0.00),v40,z0,tPen\WObj:=wPaper;
    MoveL Offs(pOrigin,206.44,293.58,0.00),v40,z0,tPen\WObj:=wPaper;
    MoveL Offs(pOrigin,204.74,292.73,0.00),v40,z0,tPen\WObj:=wPaper;
    MoveL Offs(pOrigin,203.25,291.45,0.00),v40,z0,tPen\WObj:=wPaper;
    MoveL Offs(pOrigin,202.40,290.17,0.00),v40,z0,tPen\WObj:=wPaper;
    MoveL Offs(pOrigin,201.69,289.75,0.00),v40,z0,tPen\WObj:=wPaper;
    MoveL Offs(pOrigin,201.55,288.69,0.00),v40,fine,tPen\WObj:=wPaper;
    MoveL Offs(pOrigin,201.55,288.69,6.00),v60,z5,tPen\WObj:=wPaper;
    MoveL Offs(pOrigin,200.27,289.54,6.00),vTravel,z5,tPen\WObj:=wPaper;
    MoveL Offs(pOrigin,200.27,289.54,0.00),v60,z0,tPen\WObj:=wPaper;
    MoveL Offs(pOrigin,200.49,289.96,0.00),v40,z0,tPen\WObj:=wPaper;
    MoveL Offs(pOrigin,200.27,289.54,0.00),v40,fine,tPen\WObj:=wPaper;
    MoveL Offs(pOrigin,200.27,289.54,6.00),v60,z5,tPen\WObj:=wPaper;
    MoveL Offs(pOrigin,203.68,286.14,6.00),vTravel,z5,tPen\WObj:=wPaper;
    MoveL Offs(pOrigin,203.68,286.14,0.00),v60,z0,tPen\WObj:=wPaper;
    MoveL Offs(pOrigin,202.61,285.92,0.00),v40,z0,tPen\WObj:=wPaper;
    MoveL Offs(pOrigin,200.27,281.67,0.00),v40,z0,tPen\WObj:=wPaper;
    MoveL Offs(pOrigin,200.27,281.67,0.00),v40,z0,tPen\WObj:=wPaper;
    MoveL Offs(pOrigin,199.99,280.61,0.00),v40,z0,tPen\WObj:=wPaper;
    MoveL Offs(pOrigin,198.79,279.12,0.00),v40,z0,tPen\WObj:=wPaper;
    MoveL Offs(pOrigin,196.45,278.06,0.00),v40,z0,tPen\WObj:=wPaper;
    MoveL Offs(pOrigin,197.30,278.70,0.00),v40,z0,tPen\WObj:=wPaper;
    MoveL Offs(pOrigin,197.51,279.34,0.00),v40,z0,tPen\WObj:=wPaper;
    MoveL Offs(pOrigin,199.21,281.25,0.00),v40,z0,tPen\WObj:=wPaper;
    MoveL Offs(pOrigin,200.27,281.67,0.00),v40,fine,tPen\WObj:=wPaper;
    MoveL Offs(pOrigin,200.27,281.67,6.00),v60,z5,tPen\WObj:=wPaper;
    MoveL Offs(pOrigin,198.57,280.61,6.00),vTravel,z5,tPen\WObj:=wPaper;
    MoveL Offs(pOrigin,198.57,280.61,0.00),v60,z0,tPen\WObj:=wPaper;
    MoveL Offs(pOrigin,197.30,279.34,0.00),v40,z0,tPen\WObj:=wPaper;
    MoveL Offs(pOrigin,197.30,279.34,0.00),v40,z0,tPen\WObj:=wPaper;
    MoveL Offs(pOrigin,196.45,279.76,0.00),v40,z0,tPen\WObj:=wPaper;
    MoveL Offs(pOrigin,195.18,278.91,0.00),v40,z0,tPen\WObj:=wPaper;
    MoveL Offs(pOrigin,194.54,278.98,0.00),v40,z0,tPen\WObj:=wPaper;
    MoveL Offs(pOrigin,194.32,279.34,0.00),v40,fine,tPen\WObj:=wPaper;
    MoveL Offs(pOrigin,194.32,279.34,6.00),v60,z5,tPen\WObj:=wPaper;
    MoveL Offs(pOrigin,194.32,281.04,6.00),vTravel,z5,tPen\WObj:=wPaper;
    MoveL Offs(pOrigin,194.32,281.04,0.00),v60,z0,tPen\WObj:=wPaper;
    MoveL Offs(pOrigin,196.02,282.45,0.00),v40,z0,tPen\WObj:=wPaper;
    MoveL Offs(pOrigin,196.88,282.74,0.00),v40,z0,tPen\WObj:=wPaper;
    MoveL Offs(pOrigin,197.80,283.80,0.00),v40,z0,tPen\WObj:=wPaper;
    MoveL Offs(pOrigin,197.94,284.44,0.00),v40,fine,tPen\WObj:=wPaper;
    MoveL Offs(pOrigin,197.94,284.44,6.00),v60,z5,tPen\WObj:=wPaper;
    MoveL Offs(pOrigin,194.96,285.50,6.00),vTravel,z5,tPen\WObj:=wPaper;
    MoveL Offs(pOrigin,194.96,285.50,0.00),v60,z0,tPen\WObj:=wPaper;
    MoveL Offs(pOrigin,195.18,285.92,0.00),v40,z0,tPen\WObj:=wPaper;
    MoveL Offs(pOrigin,194.96,285.50,0.00),v40,fine,tPen\WObj:=wPaper;
    MoveL Offs(pOrigin,194.96,285.50,6.00),v60,z5,tPen\WObj:=wPaper;
    MoveL Offs(pOrigin,201.34,283.38,6.00),vTravel,z5,tPen\WObj:=wPaper;
    MoveL Offs(pOrigin,201.34,283.38,0.00),v60,z0,tPen\WObj:=wPaper;
    MoveL Offs(pOrigin,201.55,283.80,0.00),v40,z0,tPen\WObj:=wPaper;
    MoveL Offs(pOrigin,201.34,283.38,0.00),v40,fine,tPen\WObj:=wPaper;
    MoveL Offs(pOrigin,201.34,283.38,6.00),v60,z5,tPen\WObj:=wPaper;
    MoveL Offs(pOrigin,202.82,281.67,6.00),vTravel,z5,tPen\WObj:=wPaper;
    MoveL Offs(pOrigin,202.82,281.67,0.00),v60,z0,tPen\WObj:=wPaper;
    MoveL Offs(pOrigin,203.18,280.61,0.00),v40,z0,tPen\WObj:=wPaper;
    MoveL Offs(pOrigin,202.19,279.98,0.00),v40,z0,tPen\WObj:=wPaper;
    MoveL Offs(pOrigin,201.34,277.85,0.00),v40,z0,tPen\WObj:=wPaper;
    MoveL Offs(pOrigin,201.76,277.00,0.00),v40,z0,tPen\WObj:=wPaper;
    MoveL Offs(pOrigin,201.55,276.58,0.00),v40,z0,tPen\WObj:=wPaper;
    MoveL Offs(pOrigin,201.34,277.42,0.00),v40,z0,tPen\WObj:=wPaper;
    MoveL Offs(pOrigin,200.06,276.58,0.00),v40,z0,tPen\WObj:=wPaper;
    MoveL Offs(pOrigin,199.07,275.30,0.00),v40,z0,tPen\WObj:=wPaper;
    MoveL Offs(pOrigin,198.93,274.24,0.00),v40,z0,tPen\WObj:=wPaper;
    MoveL Offs(pOrigin,198.15,273.60,0.00),v40,fine,tPen\WObj:=wPaper;
    MoveL Offs(pOrigin,198.15,273.60,6.00),v60,z5,tPen\WObj:=wPaper;
    MoveL Offs(pOrigin,199.00,275.51,6.00),vTravel,z5,tPen\WObj:=wPaper;
    MoveL Offs(pOrigin,199.00,275.51,0.00),v60,z0,tPen\WObj:=wPaper;
    MoveL Offs(pOrigin,199.64,276.15,0.00),v40,z0,tPen\WObj:=wPaper;
    MoveL Offs(pOrigin,200.06,276.79,0.00),v40,z0,tPen\WObj:=wPaper;
    MoveL Offs(pOrigin,200.49,277.21,0.00),v40,z0,tPen\WObj:=wPaper;
    MoveL Offs(pOrigin,200.06,276.79,0.00),v40,fine,tPen\WObj:=wPaper;
    MoveL Offs(pOrigin,200.06,276.79,6.00),v60,z5,tPen\WObj:=wPaper;
    MoveL Offs(pOrigin,200.91,274.45,6.00),vTravel,z5,tPen\WObj:=wPaper;
    MoveL Offs(pOrigin,200.91,274.45,0.00),v60,z0,tPen\WObj:=wPaper;
    MoveL Offs(pOrigin,199.00,270.41,0.00),v40,fine,tPen\WObj:=wPaper;
    MoveL Offs(pOrigin,199.00,270.41,6.00),v60,z5,tPen\WObj:=wPaper;
    MoveL Offs(pOrigin,200.91,270.20,6.00),vTravel,z5,tPen\WObj:=wPaper;
    MoveL Offs(pOrigin,200.91,270.20,0.00),v60,z0,tPen\WObj:=wPaper;
    MoveL Offs(pOrigin,200.98,268.29,0.00),v40,z0,tPen\WObj:=wPaper;
  ENDPROC

  PROC DrawPart43()
    MoveL Offs(pOrigin,201.98,267.01,0.00),v40,z0,tPen\WObj:=wPaper;
    MoveL Offs(pOrigin,201.98,267.01,0.00),v40,z0,tPen\WObj:=wPaper;
    MoveL Offs(pOrigin,202.97,267.65,0.00),v40,z0,tPen\WObj:=wPaper;
    MoveL Offs(pOrigin,203.68,270.84,0.00),v40,z0,tPen\WObj:=wPaper;
    MoveL Offs(pOrigin,203.46,269.77,0.00),v40,z0,tPen\WObj:=wPaper;
    MoveL Offs(pOrigin,203.68,270.20,0.00),v40,z0,tPen\WObj:=wPaper;
    MoveL Offs(pOrigin,203.46,269.77,0.00),v40,fine,tPen\WObj:=wPaper;
    MoveL Offs(pOrigin,203.46,269.77,6.00),v60,z5,tPen\WObj:=wPaper;
    MoveL Offs(pOrigin,200.91,270.84,6.00),vTravel,z5,tPen\WObj:=wPaper;
    MoveL Offs(pOrigin,200.91,270.84,0.00),v60,z0,tPen\WObj:=wPaper;
    MoveL Offs(pOrigin,202.97,275.73,0.00),v40,z0,tPen\WObj:=wPaper;
    MoveL Offs(pOrigin,204.31,276.79,0.00),v40,fine,tPen\WObj:=wPaper;
    MoveL Offs(pOrigin,204.31,276.79,6.00),v60,z5,tPen\WObj:=wPaper;
    MoveL Offs(pOrigin,201.98,272.96,6.00),vTravel,z5,tPen\WObj:=wPaper;
    MoveL Offs(pOrigin,201.98,272.96,0.00),v60,z0,tPen\WObj:=wPaper;
    MoveL Offs(pOrigin,202.19,272.11,0.00),v40,z0,tPen\WObj:=wPaper;
    MoveL Offs(pOrigin,201.90,271.26,0.00),v40,z0,tPen\WObj:=wPaper;
    MoveL Offs(pOrigin,200.91,270.84,0.00),v40,fine,tPen\WObj:=wPaper;
    MoveL Offs(pOrigin,200.91,270.84,6.00),v60,z5,tPen\WObj:=wPaper;
    MoveL Offs(pOrigin,196.45,270.41,6.00),vTravel,z5,tPen\WObj:=wPaper;
    MoveL Offs(pOrigin,196.45,270.41,0.00),v60,z0,tPen\WObj:=wPaper;
    MoveL Offs(pOrigin,196.24,270.84,0.00),v40,z0,tPen\WObj:=wPaper;
    MoveL Offs(pOrigin,196.45,270.41,0.00),v40,z0,tPen\WObj:=wPaper;
    MoveL Offs(pOrigin,196.02,271.26,0.00),v40,z0,tPen\WObj:=wPaper;
    MoveL Offs(pOrigin,195.81,271.69,0.00),v40,z0,tPen\WObj:=wPaper;
    MoveL Offs(pOrigin,196.02,271.26,0.00),v40,fine,tPen\WObj:=wPaper;
    MoveL Offs(pOrigin,196.02,271.26,6.00),v60,z5,tPen\WObj:=wPaper;
    MoveL Offs(pOrigin,194.96,273.17,6.00),vTravel,z5,tPen\WObj:=wPaper;
    MoveL Offs(pOrigin,194.96,273.17,0.00),v60,z0,tPen\WObj:=wPaper;
    MoveL Offs(pOrigin,194.75,273.60,0.00),v40,z0,tPen\WObj:=wPaper;
    MoveL Offs(pOrigin,194.96,273.17,0.00),v40,fine,tPen\WObj:=wPaper;
    MoveL Offs(pOrigin,194.96,273.17,6.00),v60,z5,tPen\WObj:=wPaper;
    MoveL Offs(pOrigin,194.32,274.45,6.00),vTravel,z5,tPen\WObj:=wPaper;
    MoveL Offs(pOrigin,194.32,274.45,0.00),v60,z0,tPen\WObj:=wPaper;
    MoveL Offs(pOrigin,193.48,275.51,0.00),v40,z0,tPen\WObj:=wPaper;
    MoveL Offs(pOrigin,194.32,274.45,0.00),v40,fine,tPen\WObj:=wPaper;
    MoveL Offs(pOrigin,194.32,274.45,6.00),v60,z5,tPen\WObj:=wPaper;
    MoveL Offs(pOrigin,195.60,276.58,6.00),vTravel,z5,tPen\WObj:=wPaper;
    MoveL Offs(pOrigin,195.60,276.58,0.00),v60,z0,tPen\WObj:=wPaper;
    MoveL Offs(pOrigin,196.88,276.36,0.00),v40,fine,tPen\WObj:=wPaper;
    MoveL Offs(pOrigin,196.88,276.36,6.00),v60,z5,tPen\WObj:=wPaper;
    MoveL Offs(pOrigin,198.79,279.34,6.00),vTravel,z5,tPen\WObj:=wPaper;
    MoveL Offs(pOrigin,198.79,279.34,0.00),v60,z0,tPen\WObj:=wPaper;
    MoveL Offs(pOrigin,199.21,279.76,0.00),v40,z0,tPen\WObj:=wPaper;
    MoveL Offs(pOrigin,198.79,279.34,0.00),v40,fine,tPen\WObj:=wPaper;
    MoveL Offs(pOrigin,198.79,279.34,6.00),v60,z5,tPen\WObj:=wPaper;
    MoveL Offs(pOrigin,198.57,266.59,6.00),vTravel,z5,tPen\WObj:=wPaper;
    MoveL Offs(pOrigin,198.57,266.59,0.00),v60,z0,tPen\WObj:=wPaper;
    MoveL Offs(pOrigin,198.15,267.01,0.00),v40,z0,tPen\WObj:=wPaper;
    MoveL Offs(pOrigin,198.57,266.59,0.00),v40,fine,tPen\WObj:=wPaper;
    MoveL Offs(pOrigin,198.57,266.59,6.00),v60,z5,tPen\WObj:=wPaper;
    MoveL Offs(pOrigin,197.30,263.83,6.00),vTravel,z5,tPen\WObj:=wPaper;
    MoveL Offs(pOrigin,197.30,263.83,0.00),v60,z0,tPen\WObj:=wPaper;
    MoveL Offs(pOrigin,197.94,264.25,0.00),v40,z0,tPen\WObj:=wPaper;
    MoveL Offs(pOrigin,197.30,263.83,0.00),v40,fine,tPen\WObj:=wPaper;
    MoveL Offs(pOrigin,197.30,263.83,6.00),v60,z5,tPen\WObj:=wPaper;
    MoveL Offs(pOrigin,198.15,262.76,6.00),vTravel,z5,tPen\WObj:=wPaper;
    MoveL Offs(pOrigin,198.15,262.76,0.00),v60,z0,tPen\WObj:=wPaper;
    MoveL Offs(pOrigin,198.57,262.98,0.00),v40,z0,tPen\WObj:=wPaper;
    MoveL Offs(pOrigin,198.15,262.76,0.00),v40,fine,tPen\WObj:=wPaper;
    MoveL Offs(pOrigin,198.15,262.76,6.00),v60,z5,tPen\WObj:=wPaper;
    MoveL Offs(pOrigin,197.30,261.70,6.00),vTravel,z5,tPen\WObj:=wPaper;
    MoveL Offs(pOrigin,197.30,261.70,0.00),v60,z0,tPen\WObj:=wPaper;
    MoveL Offs(pOrigin,197.51,262.12,0.00),v40,z0,tPen\WObj:=wPaper;
    MoveL Offs(pOrigin,197.30,261.70,0.00),v40,fine,tPen\WObj:=wPaper;
    MoveL Offs(pOrigin,197.30,261.70,6.00),v60,z5,tPen\WObj:=wPaper;
    MoveL Offs(pOrigin,196.24,262.76,6.00),vTravel,z5,tPen\WObj:=wPaper;
    MoveL Offs(pOrigin,196.24,262.76,0.00),v60,z0,tPen\WObj:=wPaper;
    MoveL Offs(pOrigin,197.09,263.61,0.00),v40,z0,tPen\WObj:=wPaper;
    MoveL Offs(pOrigin,196.24,262.76,0.00),v40,fine,tPen\WObj:=wPaper;
    MoveL Offs(pOrigin,196.24,262.76,6.00),v60,z5,tPen\WObj:=wPaper;
    MoveL Offs(pOrigin,195.60,261.70,6.00),vTravel,z5,tPen\WObj:=wPaper;
    MoveL Offs(pOrigin,195.60,261.70,0.00),v60,z0,tPen\WObj:=wPaper;
    MoveL Offs(pOrigin,195.81,262.12,0.00),v40,z0,tPen\WObj:=wPaper;
    MoveL Offs(pOrigin,195.60,261.70,0.00),v40,fine,tPen\WObj:=wPaper;
    MoveL Offs(pOrigin,195.60,261.70,6.00),v60,z5,tPen\WObj:=wPaper;
    MoveL Offs(pOrigin,198.57,260.00,6.00),vTravel,z5,tPen\WObj:=wPaper;
    MoveL Offs(pOrigin,198.57,260.00,0.00),v60,z0,tPen\WObj:=wPaper;
    MoveL Offs(pOrigin,198.79,259.22,0.00),v40,z0,tPen\WObj:=wPaper;
    MoveL Offs(pOrigin,200.84,259.79,0.00),v40,z0,tPen\WObj:=wPaper;
    MoveL Offs(pOrigin,200.63,260.35,0.00),v40,z0,tPen\WObj:=wPaper;
    MoveL Offs(pOrigin,199.85,260.64,0.00),v40,z0,tPen\WObj:=wPaper;
    MoveL Offs(pOrigin,199.00,260.50,0.00),v40,z0,tPen\WObj:=wPaper;
    MoveL Offs(pOrigin,198.57,260.00,0.00),v40,z0,tPen\WObj:=wPaper;
    MoveL Offs(pOrigin,198.57,259.15,0.00),v40,z0,tPen\WObj:=wPaper;
    MoveL Offs(pOrigin,198.15,257.24,0.00),v40,z0,tPen\WObj:=wPaper;
    MoveL Offs(pOrigin,198.36,253.84,0.00),v40,z0,tPen\WObj:=wPaper;
    MoveL Offs(pOrigin,199.99,250.23,0.00),v40,z0,tPen\WObj:=wPaper;
    MoveL Offs(pOrigin,201.12,249.59,0.00),v40,z0,tPen\WObj:=wPaper;
    MoveL Offs(pOrigin,201.12,249.59,0.00),v40,z0,tPen\WObj:=wPaper;
    MoveL Offs(pOrigin,202.97,243.85,0.00),v40,z0,tPen\WObj:=wPaper;
    MoveL Offs(pOrigin,205.80,238.32,0.00),v40,fine,tPen\WObj:=wPaper;
    MoveL Offs(pOrigin,205.80,238.32,6.00),v60,z5,tPen\WObj:=wPaper;
    MoveL Offs(pOrigin,206.65,241.51,6.00),vTravel,z5,tPen\WObj:=wPaper;
    MoveL Offs(pOrigin,206.65,241.51,0.00),v60,z0,tPen\WObj:=wPaper;
    MoveL Offs(pOrigin,207.29,233.65,0.00),v40,z0,tPen\WObj:=wPaper;
    MoveL Offs(pOrigin,207.29,233.65,0.00),v40,z0,tPen\WObj:=wPaper;
    MoveL Offs(pOrigin,207.93,233.23,0.00),v40,z0,tPen\WObj:=wPaper;
    MoveL Offs(pOrigin,207.93,232.38,0.00),v40,z0,tPen\WObj:=wPaper;
    MoveL Offs(pOrigin,207.93,232.38,0.00),v40,z0,tPen\WObj:=wPaper;
    MoveL Offs(pOrigin,209.98,225.57,0.00),v40,z0,tPen\WObj:=wPaper;
    MoveL Offs(pOrigin,211.89,221.75,0.00),v40,z0,tPen\WObj:=wPaper;
    MoveL Offs(pOrigin,215.15,217.29,0.00),v40,z0,tPen\WObj:=wPaper;
    MoveL Offs(pOrigin,222.16,210.98,0.00),v40,z0,tPen\WObj:=wPaper;
    MoveL Offs(pOrigin,227.90,208.72,0.00),v40,z0,tPen\WObj:=wPaper;
    MoveL Offs(pOrigin,229.81,208.36,0.00),v40,fine,tPen\WObj:=wPaper;
    MoveL Offs(pOrigin,229.81,208.36,6.00),v60,z5,tPen\WObj:=wPaper;
    MoveL Offs(pOrigin,226.13,205.74,6.00),vTravel,z5,tPen\WObj:=wPaper;
    MoveL Offs(pOrigin,226.13,205.74,0.00),v60,z0,tPen\WObj:=wPaper;
    MoveL Offs(pOrigin,222.80,209.00,0.00),v40,z0,tPen\WObj:=wPaper;
    MoveL Offs(pOrigin,226.13,205.74,0.00),v40,fine,tPen\WObj:=wPaper;
    MoveL Offs(pOrigin,226.13,205.74,6.00),v60,z5,tPen\WObj:=wPaper;
    MoveL Offs(pOrigin,225.14,204.75,6.00),vTravel,z5,tPen\WObj:=wPaper;
    MoveL Offs(pOrigin,225.14,204.75,0.00),v60,z0,tPen\WObj:=wPaper;
    MoveL Offs(pOrigin,224.71,205.39,0.00),v40,z0,tPen\WObj:=wPaper;
    MoveL Offs(pOrigin,225.14,204.75,0.00),v40,fine,tPen\WObj:=wPaper;
    MoveL Offs(pOrigin,225.14,204.75,6.00),v60,z5,tPen\WObj:=wPaper;
    MoveL Offs(pOrigin,224.43,205.74,6.00),vTravel,z5,tPen\WObj:=wPaper;
    MoveL Offs(pOrigin,224.43,205.74,0.00),v60,z0,tPen\WObj:=wPaper;
    MoveL Offs(pOrigin,222.16,207.94,0.00),v40,z0,tPen\WObj:=wPaper;
  ENDPROC

  PROC DrawPart44()
    MoveL Offs(pOrigin,224.43,205.74,0.00),v40,fine,tPen\WObj:=wPaper;
    MoveL Offs(pOrigin,224.43,205.74,6.00),v60,z5,tPen\WObj:=wPaper;
    MoveL Offs(pOrigin,225.77,203.69,6.00),vTravel,z5,tPen\WObj:=wPaper;
    MoveL Offs(pOrigin,225.77,203.69,0.00),v60,z0,tPen\WObj:=wPaper;
    MoveL Offs(pOrigin,225.56,204.11,0.00),v40,z0,tPen\WObj:=wPaper;
    MoveL Offs(pOrigin,225.77,203.69,0.00),v40,fine,tPen\WObj:=wPaper;
    MoveL Offs(pOrigin,225.77,203.69,6.00),v60,z5,tPen\WObj:=wPaper;
    MoveL Offs(pOrigin,226.41,202.41,6.00),vTravel,z5,tPen\WObj:=wPaper;
    MoveL Offs(pOrigin,226.41,202.41,0.00),v60,z0,tPen\WObj:=wPaper;
    MoveL Offs(pOrigin,226.20,202.84,0.00),v40,z0,tPen\WObj:=wPaper;
    MoveL Offs(pOrigin,226.41,202.41,0.00),v40,fine,tPen\WObj:=wPaper;
    MoveL Offs(pOrigin,226.41,202.41,6.00),v60,z5,tPen\WObj:=wPaper;
    MoveL Offs(pOrigin,228.11,203.26,6.00),vTravel,z5,tPen\WObj:=wPaper;
    MoveL Offs(pOrigin,228.11,203.26,0.00),v60,z0,tPen\WObj:=wPaper;
    MoveL Offs(pOrigin,228.32,203.69,0.00),v40,z0,tPen\WObj:=wPaper;
    MoveL Offs(pOrigin,228.11,203.26,0.00),v40,z0,tPen\WObj:=wPaper;
    MoveL Offs(pOrigin,228.32,203.69,0.00),v40,z0,tPen\WObj:=wPaper;
    MoveL Offs(pOrigin,222.38,209.64,0.00),v40,z0,tPen\WObj:=wPaper;
    MoveL Offs(pOrigin,221.95,210.91,0.00),v40,fine,tPen\WObj:=wPaper;
    MoveL Offs(pOrigin,221.95,210.91,6.00),v60,z5,tPen\WObj:=wPaper;
    MoveL Offs(pOrigin,219.19,211.12,6.00),vTravel,z5,tPen\WObj:=wPaper;
    MoveL Offs(pOrigin,219.19,211.12,0.00),v60,z0,tPen\WObj:=wPaper;
    MoveL Offs(pOrigin,218.98,211.55,0.00),v40,z0,tPen\WObj:=wPaper;
    MoveL Offs(pOrigin,219.19,211.12,0.00),v40,z0,tPen\WObj:=wPaper;
    MoveL Offs(pOrigin,218.76,211.98,0.00),v40,z0,tPen\WObj:=wPaper;
    MoveL Offs(pOrigin,219.61,210.49,0.00),v40,z0,tPen\WObj:=wPaper;
    MoveL Offs(pOrigin,220.25,204.11,0.00),v40,z0,tPen\WObj:=wPaper;
    MoveL Offs(pOrigin,221.74,196.25,0.00),v40,z0,tPen\WObj:=wPaper;
    MoveL Offs(pOrigin,221.31,195.40,0.00),v40,z0,tPen\WObj:=wPaper;
    MoveL Offs(pOrigin,213.88,188.81,0.00),v40,z0,tPen\WObj:=wPaper;
    MoveL Offs(pOrigin,213.88,188.81,0.00),v40,z0,tPen\WObj:=wPaper;
    MoveL Offs(pOrigin,213.59,187.82,0.00),v40,z0,tPen\WObj:=wPaper;
    MoveL Offs(pOrigin,213.02,187.68,0.00),v40,z0,tPen\WObj:=wPaper;
    MoveL Offs(pOrigin,212.60,186.97,0.00),v40,z0,tPen\WObj:=wPaper;
    MoveL Offs(pOrigin,209.62,184.92,0.00),v40,z0,tPen\WObj:=wPaper;
    MoveL Offs(pOrigin,196.24,177.83,0.00),v40,z0,tPen\WObj:=wPaper;
    MoveL Offs(pOrigin,195.18,176.91,0.00),v40,z0,tPen\WObj:=wPaper;
    MoveL Offs(pOrigin,202.82,147.80,0.00),v40,z0,tPen\WObj:=wPaper;
    MoveL Offs(pOrigin,212.81,112.53,0.00),v40,z0,tPen\WObj:=wPaper;
    MoveL Offs(pOrigin,215.57,101.05,0.00),v40,z0,tPen\WObj:=wPaper;
    MoveL Offs(pOrigin,217.27,90.43,0.00),v40,z0,tPen\WObj:=wPaper;
    MoveL Offs(pOrigin,218.12,80.65,0.00),v40,z0,tPen\WObj:=wPaper;
    MoveL Offs(pOrigin,218.12,68.96,0.00),v40,z0,tPen\WObj:=wPaper;
    MoveL Offs(pOrigin,217.27,59.61,0.00),v40,z0,tPen\WObj:=wPaper;
    MoveL Offs(pOrigin,218.12,57.28,0.00),v40,z0,tPen\WObj:=wPaper;
    MoveL Offs(pOrigin,217.98,54.09,0.00),v40,z0,tPen\WObj:=wPaper;
    MoveL Offs(pOrigin,220.89,51.25,0.00),v40,z0,tPen\WObj:=wPaper;
    MoveL Offs(pOrigin,221.45,51.75,0.00),v40,z0,tPen\WObj:=wPaper;
    MoveL Offs(pOrigin,223.65,58.34,0.00),v40,z0,tPen\WObj:=wPaper;
    MoveL Offs(pOrigin,225.77,66.20,0.00),v40,z0,tPen\WObj:=wPaper;
    MoveL Offs(pOrigin,227.90,75.97,0.00),v40,z0,tPen\WObj:=wPaper;
    MoveL Offs(pOrigin,229.60,86.39,0.00),v40,z0,tPen\WObj:=wPaper;
    MoveL Offs(pOrigin,230.66,95.31,0.00),v40,z0,tPen\WObj:=wPaper;
    MoveL Offs(pOrigin,231.51,108.70,0.00),v40,z0,tPen\WObj:=wPaper;
    MoveL Offs(pOrigin,231.51,119.32,0.00),v40,z0,tPen\WObj:=wPaper;
    MoveL Offs(pOrigin,231.09,128.89,0.00),v40,z0,tPen\WObj:=wPaper;
    MoveL Offs(pOrigin,228.75,154.39,0.00),v40,z0,tPen\WObj:=wPaper;
    MoveL Offs(pOrigin,225.35,180.10,0.00),v40,z0,tPen\WObj:=wPaper;
    MoveL Offs(pOrigin,222.59,193.49,0.00),v40,z0,tPen\WObj:=wPaper;
    MoveL Offs(pOrigin,222.09,194.98,0.00),v40,z0,tPen\WObj:=wPaper;
    MoveL Offs(pOrigin,221.52,195.40,0.00),v40,fine,tPen\WObj:=wPaper;
    MoveL Offs(pOrigin,221.52,195.40,6.00),v60,z5,tPen\WObj:=wPaper;
    MoveL Offs(pOrigin,228.11,199.65,6.00),vTravel,z5,tPen\WObj:=wPaper;
    MoveL Offs(pOrigin,228.11,199.65,0.00),v60,z0,tPen\WObj:=wPaper;
    MoveL Offs(pOrigin,227.69,200.29,0.00),v40,z0,tPen\WObj:=wPaper;
    MoveL Offs(pOrigin,228.11,199.65,0.00),v40,fine,tPen\WObj:=wPaper;
    MoveL Offs(pOrigin,228.11,199.65,6.00),v60,z5,tPen\WObj:=wPaper;
    MoveL Offs(pOrigin,227.48,200.71,6.00),vTravel,z5,tPen\WObj:=wPaper;
    MoveL Offs(pOrigin,227.48,200.71,0.00),v60,z0,tPen\WObj:=wPaper;
    MoveL Offs(pOrigin,227.05,201.35,0.00),v40,z0,tPen\WObj:=wPaper;
    MoveL Offs(pOrigin,227.48,200.71,0.00),v40,fine,tPen\WObj:=wPaper;
    MoveL Offs(pOrigin,227.48,200.71,6.00),v60,z5,tPen\WObj:=wPaper;
    MoveL Offs(pOrigin,228.32,202.41,6.00),vTravel,z5,tPen\WObj:=wPaper;
    MoveL Offs(pOrigin,228.32,202.41,0.00),v60,z0,tPen\WObj:=wPaper;
    MoveL Offs(pOrigin,228.11,202.84,0.00),v40,z0,tPen\WObj:=wPaper;
    MoveL Offs(pOrigin,228.54,203.55,0.00),v40,z0,tPen\WObj:=wPaper;
    MoveL Offs(pOrigin,229.10,203.40,0.00),v40,z0,tPen\WObj:=wPaper;
    MoveL Offs(pOrigin,229.39,202.62,0.00),v40,z0,tPen\WObj:=wPaper;
    MoveL Offs(pOrigin,229.39,202.62,0.00),v40,z0,tPen\WObj:=wPaper;
    MoveL Offs(pOrigin,233.21,200.22,0.00),v40,z0,tPen\WObj:=wPaper;
    MoveL Offs(pOrigin,236.40,198.73,0.00),v40,z0,tPen\WObj:=wPaper;
    MoveL Offs(pOrigin,240.44,197.38,0.00),v40,z0,tPen\WObj:=wPaper;
    MoveL Offs(pOrigin,240.86,197.52,0.00),v40,fine,tPen\WObj:=wPaper;
    MoveL Offs(pOrigin,240.86,197.52,6.00),v60,z5,tPen\WObj:=wPaper;
    MoveL Offs(pOrigin,243.41,198.16,6.00),vTravel,z5,tPen\WObj:=wPaper;
    MoveL Offs(pOrigin,243.41,198.16,0.00),v60,z0,tPen\WObj:=wPaper;
    MoveL Offs(pOrigin,248.09,200.29,0.00),v40,z0,tPen\WObj:=wPaper;
    MoveL Offs(pOrigin,248.09,200.29,0.00),v40,z0,tPen\WObj:=wPaper;
    MoveL Offs(pOrigin,249.15,200.29,0.00),v40,z0,tPen\WObj:=wPaper;
    MoveL Offs(pOrigin,250.00,200.85,0.00),v40,z0,tPen\WObj:=wPaper;
    MoveL Offs(pOrigin,251.27,201.14,0.00),v40,z0,tPen\WObj:=wPaper;
    MoveL Offs(pOrigin,257.01,200.50,0.00),v40,z0,tPen\WObj:=wPaper;
    MoveL Offs(pOrigin,259.99,200.50,0.00),v40,z0,tPen\WObj:=wPaper;
    MoveL Offs(pOrigin,265.30,201.99,0.00),v40,fine,tPen\WObj:=wPaper;
    MoveL Offs(pOrigin,265.30,201.99,6.00),v60,z5,tPen\WObj:=wPaper;
    MoveL Offs(pOrigin,267.64,198.38,6.00),vTravel,z5,tPen\WObj:=wPaper;
    MoveL Offs(pOrigin,267.64,198.38,0.00),v60,z0,tPen\WObj:=wPaper;
    MoveL Offs(pOrigin,272.10,200.64,0.00),v40,z0,tPen\WObj:=wPaper;
    MoveL Offs(pOrigin,278.69,205.39,0.00),v40,z0,tPen\WObj:=wPaper;
    MoveL Offs(pOrigin,279.47,207.30,0.00),v40,z0,tPen\WObj:=wPaper;
    MoveL Offs(pOrigin,282.65,211.76,0.00),v40,z0,tPen\WObj:=wPaper;
    MoveL Offs(pOrigin,284.71,216.01,0.00),v40,z0,tPen\WObj:=wPaper;
    MoveL Offs(pOrigin,286.76,221.54,0.00),v40,z0,tPen\WObj:=wPaper;
    MoveL Offs(pOrigin,286.55,222.39,0.00),v40,z0,tPen\WObj:=wPaper;
    MoveL Offs(pOrigin,286.55,222.39,0.00),v40,z0,tPen\WObj:=wPaper;
    MoveL Offs(pOrigin,286.98,223.66,0.00),v40,z0,tPen\WObj:=wPaper;
    MoveL Offs(pOrigin,286.55,223.88,0.00),v40,z0,tPen\WObj:=wPaper;
    MoveL Offs(pOrigin,286.55,223.88,0.00),v40,z0,tPen\WObj:=wPaper;
    MoveL Offs(pOrigin,286.90,225.36,0.00),v40,z0,tPen\WObj:=wPaper;
    MoveL Offs(pOrigin,289.31,230.68,0.00),v40,z0,tPen\WObj:=wPaper;
    MoveL Offs(pOrigin,290.59,236.20,0.00),v40,z0,tPen\WObj:=wPaper;
    MoveL Offs(pOrigin,291.01,245.12,0.00),v40,z0,tPen\WObj:=wPaper;
    MoveL Offs(pOrigin,290.38,249.38,0.00),v40,z0,tPen\WObj:=wPaper;
    MoveL Offs(pOrigin,290.38,249.38,0.00),v40,z0,tPen\WObj:=wPaper;
    MoveL Offs(pOrigin,290.16,250.23,0.00),v40,z0,tPen\WObj:=wPaper;
    MoveL Offs(pOrigin,290.80,251.71,0.00),v40,z0,tPen\WObj:=wPaper;
    MoveL Offs(pOrigin,290.80,251.71,0.00),v40,z0,tPen\WObj:=wPaper;
    MoveL Offs(pOrigin,292.00,254.48,0.00),v40,z0,tPen\WObj:=wPaper;
    MoveL Offs(pOrigin,292.08,255.54,0.00),v40,z0,tPen\WObj:=wPaper;
    MoveL Offs(pOrigin,291.44,257.45,0.00),v40,z0,tPen\WObj:=wPaper;
  ENDPROC

  PROC DrawPart45()
    MoveL Offs(pOrigin,291.58,258.73,0.00),v40,z0,tPen\WObj:=wPaper;
    MoveL Offs(pOrigin,290.38,260.42,0.00),v40,z0,tPen\WObj:=wPaper;
    MoveL Offs(pOrigin,290.38,261.27,0.00),v40,z0,tPen\WObj:=wPaper;
    MoveL Offs(pOrigin,289.74,262.76,0.00),v40,z0,tPen\WObj:=wPaper;
    MoveL Offs(pOrigin,289.74,262.76,0.00),v40,z0,tPen\WObj:=wPaper;
    MoveL Offs(pOrigin,290.38,266.16,0.00),v40,z0,tPen\WObj:=wPaper;
    MoveL Offs(pOrigin,290.38,266.16,0.00),v40,z0,tPen\WObj:=wPaper;
    MoveL Offs(pOrigin,290.80,267.01,0.00),v40,z0,tPen\WObj:=wPaper;
    MoveL Offs(pOrigin,291.86,267.65,0.00),v40,z0,tPen\WObj:=wPaper;
    MoveL Offs(pOrigin,294.84,270.62,0.00),v40,z0,tPen\WObj:=wPaper;
    MoveL Offs(pOrigin,294.84,270.62,0.00),v40,z0,tPen\WObj:=wPaper;
    MoveL Offs(pOrigin,295.05,271.26,0.00),v40,z0,tPen\WObj:=wPaper;
    MoveL Offs(pOrigin,296.33,271.69,0.00),v40,z0,tPen\WObj:=wPaper;
    MoveL Offs(pOrigin,297.32,271.40,0.00),v40,z0,tPen\WObj:=wPaper;
    MoveL Offs(pOrigin,299.16,268.50,0.00),v40,z0,tPen\WObj:=wPaper;
    MoveL Offs(pOrigin,299.94,265.10,0.00),v40,z0,tPen\WObj:=wPaper;
    MoveL Offs(pOrigin,299.30,260.64,0.00),v40,z0,tPen\WObj:=wPaper;
    MoveL Offs(pOrigin,298.31,258.94,0.00),v40,z0,tPen\WObj:=wPaper;
    MoveL Offs(pOrigin,298.66,257.24,0.00),v40,z0,tPen\WObj:=wPaper;
    MoveL Offs(pOrigin,298.10,256.39,0.00),v40,z0,tPen\WObj:=wPaper;
    MoveL Offs(pOrigin,296.89,252.14,0.00),v40,z0,tPen\WObj:=wPaper;
    MoveL Offs(pOrigin,295.05,248.95,0.00),v40,fine,tPen\WObj:=wPaper;
    MoveL Offs(pOrigin,295.05,248.95,6.00),v60,z5,tPen\WObj:=wPaper;
    MoveL Offs(pOrigin,291.65,250.44,6.00),vTravel,z5,tPen\WObj:=wPaper;
    MoveL Offs(pOrigin,291.65,250.44,0.00),v60,z0,tPen\WObj:=wPaper;
    MoveL Offs(pOrigin,292.71,251.71,0.00),v40,z0,tPen\WObj:=wPaper;
    MoveL Offs(pOrigin,291.65,250.44,0.00),v40,fine,tPen\WObj:=wPaper;
    MoveL Offs(pOrigin,291.65,250.44,6.00),v60,z5,tPen\WObj:=wPaper;
    MoveL Offs(pOrigin,290.16,250.65,6.00),vTravel,z5,tPen\WObj:=wPaper;
    MoveL Offs(pOrigin,290.16,250.65,0.00),v60,z0,tPen\WObj:=wPaper;
    MoveL Offs(pOrigin,289.95,251.50,0.00),v40,z0,tPen\WObj:=wPaper;
    MoveL Offs(pOrigin,290.80,251.71,0.00),v40,z0,tPen\WObj:=wPaper;
    MoveL Offs(pOrigin,289.95,251.71,0.00),v40,z0,tPen\WObj:=wPaper;
    MoveL Offs(pOrigin,289.31,255.32,0.00),v40,fine,tPen\WObj:=wPaper;
    MoveL Offs(pOrigin,289.31,255.32,6.00),v60,z5,tPen\WObj:=wPaper;
    MoveL Offs(pOrigin,288.04,258.09,6.00),vTravel,z5,tPen\WObj:=wPaper;
    MoveL Offs(pOrigin,288.04,258.09,0.00),v60,z0,tPen\WObj:=wPaper;
    MoveL Offs(pOrigin,288.46,258.51,0.00),v40,z0,tPen\WObj:=wPaper;
    MoveL Offs(pOrigin,288.60,259.58,0.00),v40,z0,tPen\WObj:=wPaper;
    MoveL Offs(pOrigin,289.52,260.42,0.00),v40,fine,tPen\WObj:=wPaper;
    MoveL Offs(pOrigin,289.52,260.42,6.00),v60,z5,tPen\WObj:=wPaper;
    MoveL Offs(pOrigin,290.38,261.27,6.00),vTravel,z5,tPen\WObj:=wPaper;
    MoveL Offs(pOrigin,290.38,261.27,0.00),v60,z0,tPen\WObj:=wPaper;
    MoveL Offs(pOrigin,290.30,260.64,0.00),v40,z0,tPen\WObj:=wPaper;
    MoveL Offs(pOrigin,289.95,260.42,0.00),v40,z0,tPen\WObj:=wPaper;
    MoveL Offs(pOrigin,288.96,261.27,0.00),v40,z0,tPen\WObj:=wPaper;
    MoveL Offs(pOrigin,288.96,262.12,0.00),v40,z0,tPen\WObj:=wPaper;
    MoveL Offs(pOrigin,289.74,262.76,0.00),v40,fine,tPen\WObj:=wPaper;
    MoveL Offs(pOrigin,289.74,262.76,6.00),v60,z5,tPen\WObj:=wPaper;
    MoveL Offs(pOrigin,287.40,264.25,6.00),vTravel,z5,tPen\WObj:=wPaper;
    MoveL Offs(pOrigin,287.40,264.25,0.00),v60,z0,tPen\WObj:=wPaper;
    MoveL Offs(pOrigin,286.76,265.31,0.00),v40,z0,tPen\WObj:=wPaper;
    MoveL Offs(pOrigin,286.98,266.38,0.00),v40,z0,tPen\WObj:=wPaper;
    MoveL Offs(pOrigin,286.55,269.14,0.00),v40,z0,tPen\WObj:=wPaper;
    MoveL Offs(pOrigin,285.70,269.99,0.00),v40,z0,tPen\WObj:=wPaper;
    MoveL Offs(pOrigin,284.00,269.49,0.00),v40,z0,tPen\WObj:=wPaper;
    MoveL Offs(pOrigin,282.51,271.26,0.00),v40,fine,tPen\WObj:=wPaper;
    MoveL Offs(pOrigin,282.51,271.26,6.00),v60,z5,tPen\WObj:=wPaper;
    MoveL Offs(pOrigin,283.15,272.33,6.00),vTravel,z5,tPen\WObj:=wPaper;
    MoveL Offs(pOrigin,283.15,272.33,0.00),v60,z0,tPen\WObj:=wPaper;
    MoveL Offs(pOrigin,283.15,272.11,0.00),v40,z0,tPen\WObj:=wPaper;
    MoveL Offs(pOrigin,284.00,272.33,0.00),v40,z0,tPen\WObj:=wPaper;
    MoveL Offs(pOrigin,284.00,272.33,0.00),v40,z0,tPen\WObj:=wPaper;
    MoveL Offs(pOrigin,284.64,272.96,0.00),v40,z0,tPen\WObj:=wPaper;
    MoveL Offs(pOrigin,285.70,272.96,0.00),v40,z0,tPen\WObj:=wPaper;
    MoveL Offs(pOrigin,286.55,272.33,0.00),v40,z0,tPen\WObj:=wPaper;
    MoveL Offs(pOrigin,286.55,272.33,0.00),v40,z0,tPen\WObj:=wPaper;
    MoveL Offs(pOrigin,286.12,271.69,0.00),v40,z0,tPen\WObj:=wPaper;
    MoveL Offs(pOrigin,285.49,271.69,0.00),v40,fine,tPen\WObj:=wPaper;
    MoveL Offs(pOrigin,285.49,271.69,6.00),v60,z5,tPen\WObj:=wPaper;
    MoveL Offs(pOrigin,284.00,269.35,6.00),vTravel,z5,tPen\WObj:=wPaper;
    MoveL Offs(pOrigin,284.00,269.35,0.00),v60,z0,tPen\WObj:=wPaper;
    MoveL Offs(pOrigin,284.64,265.95,0.00),v40,z0,tPen\WObj:=wPaper;
    MoveL Offs(pOrigin,285.27,264.89,0.00),v40,z0,tPen\WObj:=wPaper;
    MoveL Offs(pOrigin,285.35,263.83,0.00),v40,z0,tPen\WObj:=wPaper;
    MoveL Offs(pOrigin,286.05,262.98,0.00),v40,z0,tPen\WObj:=wPaper;
    MoveL Offs(pOrigin,286.41,260.85,0.00),v40,z0,tPen\WObj:=wPaper;
    MoveL Offs(pOrigin,287.12,258.94,0.00),v40,z0,tPen\WObj:=wPaper;
    MoveL Offs(pOrigin,288.04,258.09,0.00),v40,fine,tPen\WObj:=wPaper;
    MoveL Offs(pOrigin,288.04,258.09,6.00),v60,z5,tPen\WObj:=wPaper;
    MoveL Offs(pOrigin,291.65,258.09,6.00),vTravel,z5,tPen\WObj:=wPaper;
    MoveL Offs(pOrigin,291.65,258.09,0.00),v60,z0,tPen\WObj:=wPaper;
    MoveL Offs(pOrigin,292.71,257.66,0.00),v40,z0,tPen\WObj:=wPaper;
    MoveL Offs(pOrigin,293.14,253.41,0.00),v40,z0,tPen\WObj:=wPaper;
    MoveL Offs(pOrigin,293.14,253.41,0.00),v40,z0,tPen\WObj:=wPaper;
    MoveL Offs(pOrigin,292.50,251.71,0.00),v40,z0,tPen\WObj:=wPaper;
    MoveL Offs(pOrigin,291.15,249.80,0.00),v40,z0,tPen\WObj:=wPaper;
    MoveL Offs(pOrigin,290.38,249.38,0.00),v40,fine,tPen\WObj:=wPaper;
    MoveL Offs(pOrigin,290.38,249.38,6.00),v60,z5,tPen\WObj:=wPaper;
    MoveL Offs(pOrigin,293.14,253.41,6.00),vTravel,z5,tPen\WObj:=wPaper;
    MoveL Offs(pOrigin,293.14,253.41,0.00),v60,z0,tPen\WObj:=wPaper;
    MoveL Offs(pOrigin,293.77,253.48,0.00),v40,z0,tPen\WObj:=wPaper;
    MoveL Offs(pOrigin,294.27,254.26,0.00),v40,z0,tPen\WObj:=wPaper;
    MoveL Offs(pOrigin,294.84,257.88,0.00),v40,fine,tPen\WObj:=wPaper;
    MoveL Offs(pOrigin,294.84,257.88,6.00),v60,z5,tPen\WObj:=wPaper;
    MoveL Offs(pOrigin,298.02,256.60,6.00),vTravel,z5,tPen\WObj:=wPaper;
    MoveL Offs(pOrigin,298.02,256.60,0.00),v60,z0,tPen\WObj:=wPaper;
    MoveL Offs(pOrigin,297.81,258.09,0.00),v40,z0,tPen\WObj:=wPaper;
    MoveL Offs(pOrigin,298.24,258.51,0.00),v40,fine,tPen\WObj:=wPaper;
    MoveL Offs(pOrigin,298.24,258.51,6.00),v60,z5,tPen\WObj:=wPaper;
    MoveL Offs(pOrigin,298.45,259.79,6.00),vTravel,z5,tPen\WObj:=wPaper;
    MoveL Offs(pOrigin,298.45,259.79,0.00),v60,z0,tPen\WObj:=wPaper;
    MoveL Offs(pOrigin,297.95,260.21,0.00),v40,z0,tPen\WObj:=wPaper;
    MoveL Offs(pOrigin,295.69,268.08,0.00),v40,fine,tPen\WObj:=wPaper;
    MoveL Offs(pOrigin,295.69,268.08,6.00),v60,z5,tPen\WObj:=wPaper;
    MoveL Offs(pOrigin,294.84,270.62,6.00),vTravel,z5,tPen\WObj:=wPaper;
    MoveL Offs(pOrigin,294.84,270.62,0.00),v60,z0,tPen\WObj:=wPaper;
    MoveL Offs(pOrigin,297.60,270.62,0.00),v40,fine,tPen\WObj:=wPaper;
    MoveL Offs(pOrigin,297.60,270.62,6.00),v60,z5,tPen\WObj:=wPaper;
    MoveL Offs(pOrigin,299.73,271.69,6.00),vTravel,z5,tPen\WObj:=wPaper;
    MoveL Offs(pOrigin,299.73,271.69,0.00),v60,z0,tPen\WObj:=wPaper;
    MoveL Offs(pOrigin,299.30,272.33,0.00),v40,z0,tPen\WObj:=wPaper;
    MoveL Offs(pOrigin,299.73,271.69,0.00),v40,z0,tPen\WObj:=wPaper;
    MoveL Offs(pOrigin,299.09,272.54,0.00),v40,z0,tPen\WObj:=wPaper;
    MoveL Offs(pOrigin,298.24,273.39,0.00),v40,z0,tPen\WObj:=wPaper;
    MoveL Offs(pOrigin,299.09,272.54,0.00),v40,fine,tPen\WObj:=wPaper;
    MoveL Offs(pOrigin,299.09,272.54,6.00),v60,z5,tPen\WObj:=wPaper;
    MoveL Offs(pOrigin,300.79,272.54,6.00),vTravel,z5,tPen\WObj:=wPaper;
    MoveL Offs(pOrigin,300.79,272.54,0.00),v60,z0,tPen\WObj:=wPaper;
    MoveL Offs(pOrigin,300.36,273.17,0.00),v40,z0,tPen\WObj:=wPaper;
  ENDPROC

